// TIA Portal V20 export
FUNCTION_BLOCK "CallUnit"   // FB130, LAD
TITLE = CallUnit
// This block calls all functionality inside the unit.
// stored: IsIECCheckEnabled true, MemoryReserve 100, Namespace Unit1, SetENOAutomatically true
   VAR_INPUT
      safetyReleased : Bool;   // Status from safety program
   END_VAR
   VAR_OUTPUT
      acknowledgeSafety { ExternalWritable := 'False'} : Bool;   // Acknowledge command to the safety program
   END_VAR
   VAR_IN_OUT
      globalStatus : "LAF_typeGeneralStatus";   // Global status
      unitInterface : "LAF_typeUnitInterface";   // Global unit interface
   END_VAR
   VAR
      instManageAlarms { ExternalWritable := 'False'} : "LAF_ManageAlarms";
      instStatusCollector { ExternalWritable := 'False'} : "LUC_StatusCollector";
      instInterfaceManager { ExternalWritable := 'False'} : "LUC_InterfaceManager";
      instUnitModeStateManager { ExternalWritable := 'False'} : "LPMLV2022_UnitModeStateManager";
      instRemoteInterfaceOpcUa { ExternalWritable := 'False'} : "LUC_RemoteCtrl_OpcUa";
      instSignalStack { ExternalWritable := 'False'} : "LUC_SignalStack";
      instUnitModeStateTimes { ExternalWritable := 'False'} : "LPMLV2022_UnitModeStateTimes";
      instUnitModeChangeAllowed { ExternalWritable := 'False'} : "LPMLV2022_UnitModeChangeAllowed";
      instPFEEvents { ExternalWritable := 'False'} : "Unit1.EventsPFE";
      instTonTimer { ExternalWritable := 'False'} : Array[0..9] of TON_TIME;
      instTofTimer { ExternalWritable := 'False'} : Array[0..9] of TOF_TIME;
      instEQP_Interface_BA030 { ExternalWritable := 'False'} : "LER_EQP_Interface";
      instEQP_Interface_BA040 { ExternalWritable := 'False'} : "LER_EQP_Interface";
      instSinaInfeed { ExternalWritable := 'False'} : SinaInfeed;
      instLER_FFU_LIU117 { ExternalWritable := 'False'} : "LER_FFU_LIU117";
      statRemoteInterface { ExternalWritable := 'False'} : "LUC_typeCommands";
      statLocalInterface { ExternalWritable := 'False'} : "LUC_typeCommands";
      statEmEnableCheck { ExternalWritable := 'False'} : Array[0..2] of Bool;
      statEmHomedCheck { ExternalWritable := 'False'} : Array[0..2] of Bool;
      statPulse { ExternalWritable := 'False'} : Array[0..99] of Bool;
      statCycleTime { ExternalWritable := 'False'} : Struct
         Buffer1 : LReal;
         Buffer2 : DInt;
         Buffer3 : DInt;
         Buffer4 : DInt;
         Buffer5 : DInt;
      END_STRUCT;
      statEnableManualCmds : Bool;
      statAllEmLinked { ExternalWritable := 'False'} : Bool;
      citi_Ptrig : Array[0..20] of Bool;
      citiTon : Array[0..20] of TON_TIME;
      citi : Time;
      citiTest : Array[0..20] of Bool;
   END_VAR
   VAR_TEMP
      tempUnitFeedback : "LUC_typeStateCommands";   // Collected commands in the unit, e.g. direct command or commands derived from alarms
      tempProcessCommands : "LUC_typeStateCommands";   // Requested unit state changes by the process
      tempUnitMode : DInt;   // Requested unit mode
      tempUnitModeChangeRequest : Bool;   // Request unit mode
      tempCntrlCmd : DInt;   // Request control command
      tempCmdChangeRequest : Bool;   // Enable change into requested state
      tempSc : Bool;   // State change from FALSE to TRUE (rising edge) triggers state complete signal
      tempPartData : "LER_typePartData";
      tempPartData_All : Array[0..18] of "LER_typePartData";
      tempTimeMs : DInt;
   END_VAR
   VAR CONSTANT
      TRUE : Bool := TRUE;
      FALSE : Bool := FALSE;
   END_VAR
   VAR_TEMP   // added for the SCL form of the ladder/FBD networks
      _w1 : Bool;
      _w2 : Bool;
      _w3 : Bool;
      _w4 : Bool;
      _w5 : Bool;
      _w6 : Bool;
      _w7 : Bool;
      _w8 : Bool;
   END_VAR
BEGIN

REGION Network 1: BLOCK INFO HEADER
   // (company) / (C) Copyright (year)
   // ---------------------------------------------------------------------------------
   // Title:                             (Title of this block)
   // Comment/Function: (that is implemented in the block)
   // Library/Family:           (that the source is dedicated to)
   // Author:                        (department / person in charge / contact)
   // Target System:          (test system with FW version)
   // Engineering:              TIA Portal (SW version)
   // Restrictions:               (OB types, etc.)
   // Requirements:           (hardware, technological package, etc.)
   // ---------------------------------------------------------------------------------
   // Change log table:
   // Version          | Date             | Signature      | Expert in charge  | Changes applied ------------------------|----------------------|-------------------------|--------------------------------|-----------------------
   // 001.000.000 | yyyy-mm-dd | 0x00000000 | (name of expert) | First released version
END_REGION

REGION Network 2: DESCRIPTION
   // This is a template block provided by the Automation Framework. It can be used to create an own project.
   // The Block Info Header is prepared to put in your own data.
   // Description of the block could be added here and the docu created by Code2Docu.
END_REGION

REGION Network 3: Simulation
   // If simulation is active on a global level, inherit this status and set simulation active in this unit also. Information is written to DB ControlNodes, from where it is distributed to the equipmemt modules.
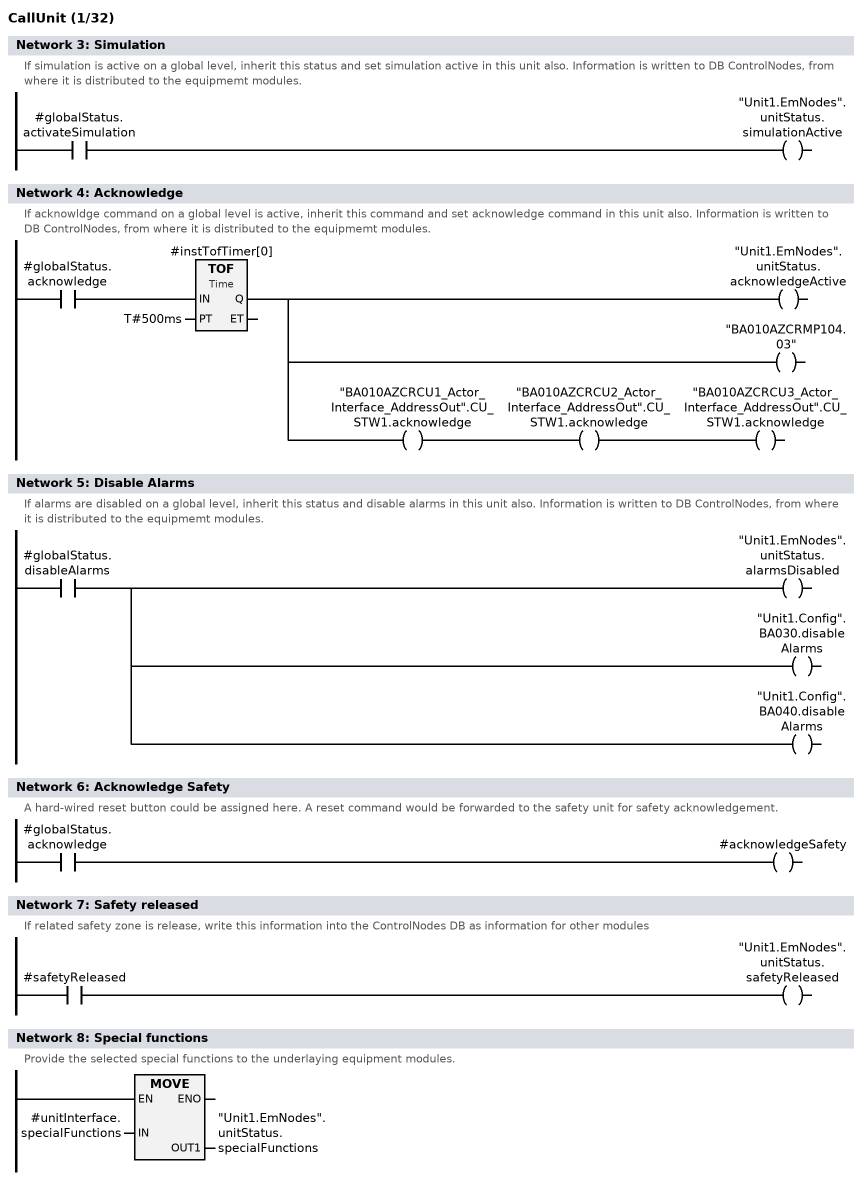
   RUNG wire#powerrail
      Contact( #globalStatus.activateSimulation )
      Coil( "Unit1.EmNodes".unitStatus.simulationActive )
   END_RUNG
   // the same network as SCL:
   "Unit1.EmNodes".unitStatus.simulationActive := #globalStatus.activateSimulation;
END_REGION

REGION Network 4: Acknowledge
   // If acknowldge command on a global level is active, inherit this command and set acknowledge command in this unit also. Information is written to DB ControlNodes, from where it is distributed to the equipmemt modules.
   RUNG wire#powerrail
      Contact( #globalStatus.acknowledge )
      { S7_Templates := "time_type := Time" } #instTofTimer[0].TOF(pt := T#500ms, et =>)
      wire#w1
      Coil( "Unit1.EmNodes".unitStatus.acknowledgeActive )
   END_RUNG
   RUNG wire#w1
      Coil( "BA010AZCRMP104.03" )
   END_RUNG
   RUNG wire#w1
      Coil( "BA010AZCRCU1_Actor_Interface_AddressOut".CU_STW1.acknowledge )
      Coil( "BA010AZCRCU2_Actor_Interface_AddressOut".CU_STW1.acknowledge )
      Coil( "BA010AZCRCU3_Actor_Interface_AddressOut".CU_STW1.acknowledge )
   END_RUNG
   // the same network as SCL:
   #instTofTimer[0].TOF(IN := #globalStatus.acknowledge, PT := T#500ms);
   "Unit1.EmNodes".unitStatus.acknowledgeActive := #instTofTimer[0].Q;
   "BA010AZCRMP104.03" := #instTofTimer[0].Q;
   "BA010AZCRCU1_Actor_Interface_AddressOut".CU_STW1.acknowledge := #instTofTimer[0].Q;
   "BA010AZCRCU2_Actor_Interface_AddressOut".CU_STW1.acknowledge := #instTofTimer[0].Q;
   "BA010AZCRCU3_Actor_Interface_AddressOut".CU_STW1.acknowledge := #instTofTimer[0].Q;
END_REGION

REGION Network 5: Disable Alarms
   // If alarms are disabled on a global level, inherit this status and disable alarms in this unit also. Information is written to DB ControlNodes, from where it is distributed to the equipmemt modules.
   RUNG wire#powerrail
      Contact( #globalStatus.disableAlarms )
      wire#w1
      Coil( "Unit1.EmNodes".unitStatus.alarmsDisabled )
   END_RUNG
   RUNG wire#w1
      Coil( "Unit1.Config".BA030.disableAlarms )
   END_RUNG
   RUNG wire#w1
      Coil( "Unit1.Config".BA040.disableAlarms )
   END_RUNG
   // the same network as SCL:
   "Unit1.EmNodes".unitStatus.alarmsDisabled := #globalStatus.disableAlarms;
   "Unit1.Config".BA030.disableAlarms := #globalStatus.disableAlarms;
   "Unit1.Config".BA040.disableAlarms := #globalStatus.disableAlarms;
END_REGION

REGION Network 6: Acknowledge Safety
   // A hard-wired reset button could be assigned here. A reset command would be forwarded to the safety unit for safety acknowledgement.
   RUNG wire#powerrail
      Contact( #globalStatus.acknowledge )
      Coil( #acknowledgeSafety )
   END_RUNG
   // the same network as SCL:
   #acknowledgeSafety := #globalStatus.acknowledge;
END_REGION

REGION Network 7: Safety released
   // If related safety zone is release, write this information into the ControlNodes DB as information for other modules
   RUNG wire#powerrail
      Contact( #safetyReleased )
      Coil( "Unit1.EmNodes".unitStatus.safetyReleased )
   END_RUNG
   // the same network as SCL:
   "Unit1.EmNodes".unitStatus.safetyReleased := #safetyReleased;
END_REGION

REGION Network 8: Special functions
   // Provide the selected special functions to the underlaying equipment modules.
   RUNG wire#powerrail
      Move(in := #unitInterface.specialFunctions, out1 => "Unit1.EmNodes".unitStatus.specialFunctions)
   END_RUNG
   // the same network as SCL:
   "Unit1.EmNodes".unitStatus.specialFunctions := #unitInterface.specialFunctions;
END_REGION

REGION Network 9 (SCL): Electric Power CB
   // E.g. put the feedback of circuit breakers or power supplies here.
   // DC24 Voltage
   "Unit1.ControlNodes".fuses.E726CbVoltage24VOK := "BA010AZCRMP101.12";
   "Unit1.ControlNodes".fuses.E4304CbVoltage24VOK := "BA010AZCRMP101.17";
   "Unit1.ControlNodes".fuses.E4420CbVoltage24VOK := "BA010AZCRMP101.22";
   "Unit1.ControlNodes".fuses.E4426CbVoltage24VOK := "BA010AZCRMP101.23";
   "Unit1.ControlNodes".fuses.E4432CbVoltage24VOK := "BA010AZCRMP101.24";
   "Unit1.ControlNodes".fuses.E4456CbVoltage24VOK := "BA010AZCRMP101.25";
   "Unit1.ControlNodes".fuses.E5110CbVoltage24VOK := "BA010AZCRMP101.31";
   "Unit1.ControlNodes".fuses.E5116CbVoltage24VOK := "BA010AZCRMP101.32";
   "Unit1.ControlNodes".fuses.E5160CbVoltage24VOK := "BA010AZCRMP101.33";
   "Unit1.ControlNodes".fuses.E5166CbVoltage24VOK := "BA010AZCRMP101.34";
   "Unit1.ControlNodes".fuses.E5172CbVoltage24VOK := "BA010AZCRMP101.35";
   "Unit1.ControlNodes".fuses.E5222CbVoltage24VOK := "BA010AZCRMP101.37";
   "Unit1.ControlNodes".fuses.E6154CbVoltage24VOK := "BA010AZCRMP102.02";
   "Unit1.ControlNodes".fuses.E6180CbVoltage24VOK := "BA010AZCRMP102.03";
   "Unit1.ControlNodes".fuses.E6204CbVoltage24VOK := "BA010AZCRMP102.04";
   "Unit1.ControlNodes".fuses.E6206CbVoltage24VOK := "BA010AZCRMP102.05";
   "Unit1.ControlNodes".fuses.E6220CbVoltage24VOK := "BA010AZCRMP102.06";
   "Unit1.ControlNodes".fuses.E6224CbVoltage24VOK := "BA010AZCRMP102.07";
   "Unit1.ControlNodes".fuses.E6228CbVoltage24VOK := "BA010AZCRMP102.10";
   "Unit1.ControlNodes".fuses.E6304CbVoltage24VOK := "BA010AZCRMP102.12";
   "Unit1.ControlNodes".fuses.E6406CbVoltage24VOK := "BA010AZCRMP102.15";
   "Unit1.ControlNodes".fuses.E6416CbVoltage24VOK := "BA010AZCRMP102.16";
   "Unit1.ControlNodes".fuses.E6422CbVoltage24VOK := "BA010AZCRMP102.17";
   "Unit1.ControlNodes".fuses.E6456CbVoltage24VOK := "BA010AZCRMP102.21";
   "Unit1.ControlNodes".fuses.E6462CbVoltage24VOK := "BA010AZCRMP102.22";
   "Unit1.ControlNodes".fuses.E6468CbVoltage24VOK := "BA010AZCRMP102.23";
   "Unit1.ControlNodes".fuses.E6706CbVoltage24VOK := "BA010AZCRMP102.27";
   "Unit1.ControlNodes".fuses.E6716CbVoltage24VOK := "BA010AZCRMP102.30";
   "Unit1.ControlNodes".fuses.E6722CbVoltage24VOK := "BA010AZCRMP102.31";
   "Unit1.ControlNodes".fuses.E6728CbVoltage24VOK := "BA010AZCRMP102.32";
   "Unit1.ControlNodes".fuses.E6734CbVoltage24VOK := "BA010AZCRMP102.33";
   "Unit1.ControlNodes".fuses.E6756CbVoltage24VOK := "BA010AZCRMP102.34";
   "Unit1.ControlNodes".fuses.E6762CbVoltage24VOK := "BA010AZCRMP102.35";
   "Unit1.ControlNodes".fuses.E6768CbVoltage24VOK := "BA010AZCRMP102.36";
   "Unit1.ControlNodes".fuses.E6774CbVoltage24VOK := "BA010AZCRMP102.37";
   "Unit1.ControlNodes".fuses.E6780CbVoltage24VOK := "BA010AZCRMP103.00";
   "Unit1.ControlNodes".fuses.E6786CbVoltage24VOK := "BA010AZCRMP103.01";
   "Unit1.ControlNodes".fuses.E6806CbVoltage24VOK := "BA010AZCRMP103.03";
   "Unit1.ControlNodes".fuses.E6816CbVoltage24VOK := "BA010AZCRMP103.04";
   "Unit1.ControlNodes".fuses.E6836CbVoltage24VOK := "BA010AZCRMP103.05";
   "Unit1.ControlNodes".fuses.E6856CbVoltage24VOK := "BA010AZCRMP103.06";
   "Unit1.ControlNodes".fuses.E110CbVoltage24VOK := "BA010AZCRSP201.10";
   "Unit1.ControlNodes".fuses.E156CbVoltage24VOK := "BA010AZCRSP501.00";
   "Unit1.ControlNodes".fuses.E218CbVoltage24VOK := "BA010AZCRSP501.01";

   // AC480 Voltage
   "Unit1.ControlNodes".fuses.E202Cb480vVoltage24VOK := "BA010AZCRMP101.00";
   "Unit1.ControlNodes".fuses.E208Cb480vVoltage24VOK := "BA010AZCRMP101.01";
   "Unit1.ControlNodes".fuses.E214Cb480vVoltage24VOK := "BA010AZCRMP101.02";
   "Unit1.ControlNodes".fuses.E220Cb480vVoltage24VOK := "BA010AZCRMP101.03";
   "Unit1.ControlNodes".fuses.E320Cb480vVoltage24VOK := "BA010AZCRMP101.05";
   "Unit1.ControlNodes".fuses.E326Cb480vVoltage24VOK := "BA010AZCRMP101.06";
   "Unit1.ControlNodes".fuses.E332Cb480vVoltage24VOK := "BA010AZCRMP101.07";
   "Unit1.ControlNodes".fuses.E720Cb480vVoltage24VOK := "BA010AZCRMP101.11";
   "Unit1.ControlNodes".fuses.E4116Cb480vVoltage24VOK := "BA010AZCRMP101.14";
   "Unit1.ControlNodes".fuses.E4156Cb480vVoltage24VOK := "BA010AZCRMP101.15";
   "Unit1.ControlNodes".fuses.E5100Cb480vVoltage24VOK := "BA010AZCRMP101.30";
END_REGION

REGION Network 10 (SCL): Power Supply
   "Unit1.ControlNodes".pws.powerSupplyE4404PwsOK := "BA010AZCRMP101.21";
   "Unit1.ControlNodes".pws.powerSupplyE6104PwsOK := "BA010AZCRMP102.01";
   "Unit1.ControlNodes".pws.powerSupplyE6404PwsOK := "BA010AZCRMP102.14";
   "Unit1.ControlNodes".pws.powerSupplyE6704PwsOK := "BA010AZCRMP102.26";
   "Unit1.ControlNodes".pws.powerSupplyE6804PwsOK := "BA010AZCRMP103.02";
END_REGION

REGION Network 11: Main Air OK
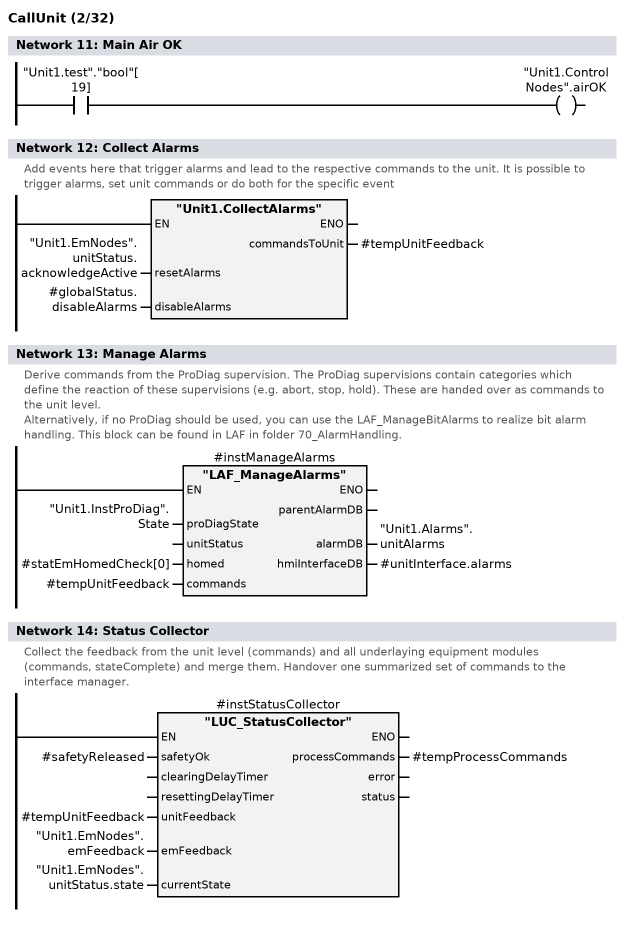
   RUNG wire#powerrail
      Contact( "Unit1.test"."bool"[19] )
      Coil( "Unit1.ControlNodes".airOK )
   END_RUNG
   // the same network as SCL:
   "Unit1.ControlNodes".airOK := "Unit1.test"."bool"[19];
END_REGION

REGION Network 12: Collect Alarms
   // Add events here that trigger alarms and lead to the respective commands to the unit. It is possible to trigger alarms, set unit commands or do both for the specific event
   RUNG wire#powerrail
      "Unit1.CollectAlarms"(resetAlarms := "Unit1.EmNodes".unitStatus.acknowledgeActive, disableAlarms := #globalStatus.disableAlarms, commandsToUnit => #tempUnitFeedback)
   END_RUNG
   // the same network as SCL:
   "Unit1.CollectAlarms"(resetAlarms := "Unit1.EmNodes".unitStatus.acknowledgeActive,
                         disableAlarms := #globalStatus.disableAlarms,
                         commandsToUnit => #tempUnitFeedback);
END_REGION

REGION Network 13: Manage Alarms
   // Derive commands from the ProDiag supervision. The ProDiag supervisions contain categories which define the reaction of these supervisions (e.g. abort, stop, hold). These are handed over as commands to the unit level.
   // Alternatively, if no ProDiag should be used, you can use the LAF_ManageBitAlarms to realize bit alarm handling. This block can be found in LAF in folder 70_AlarmHandling.
   RUNG wire#powerrail
      #instManageAlarms(proDiagState := "Unit1.InstProDiag".State, unitStatus :=, homed := #statEmHomedCheck[0], commands := #tempUnitFeedback, parentAlarmDB =>, alarmDB => "Unit1.Alarms".unitAlarms, hmiInterfaceDB => #unitInterface.alarms)
   END_RUNG
   // the same network as SCL:
   #instManageAlarms(proDiagState := "Unit1.InstProDiag".State,   // "LAF_ManageAlarms"
                     homed := #statEmHomedCheck[0],
                     commands := #tempUnitFeedback,
                     alarmDB => "Unit1.Alarms".unitAlarms,
                     hmiInterfaceDB => #unitInterface.alarms);
END_REGION

REGION Network 14: Status Collector
   // Collect the feedback from the unit level (commands) and all underlaying equipment modules (commands, stateComplete) and merge them. Handover one summarized set of commands to the interface manager.
   RUNG wire#powerrail
      #instStatusCollector(safetyOk := #safetyReleased, clearingDelayTimer :=, resettingDelayTimer :=, unitFeedback := #tempUnitFeedback, emFeedback := "Unit1.EmNodes".emFeedback, currentState := "Unit1.EmNodes".unitStatus.state, processCommands => #tempProcessCommands, error =>, status =>)
   END_RUNG
   // the same network as SCL:
   #instStatusCollector(safetyOk := #safetyReleased,   // "LUC_StatusCollector"
                        unitFeedback := #tempUnitFeedback,
                        emFeedback := "Unit1.EmNodes".emFeedback,
                        currentState := "Unit1.EmNodes".unitStatus.state,
                        processCommands => #tempProcessCommands);
END_REGION

REGION Network 15: Interface Manager
   // Read the commands from all interfaces (process, local, hmi, remote) and merge them. Handover one summarized set of commands to the mode state manager.
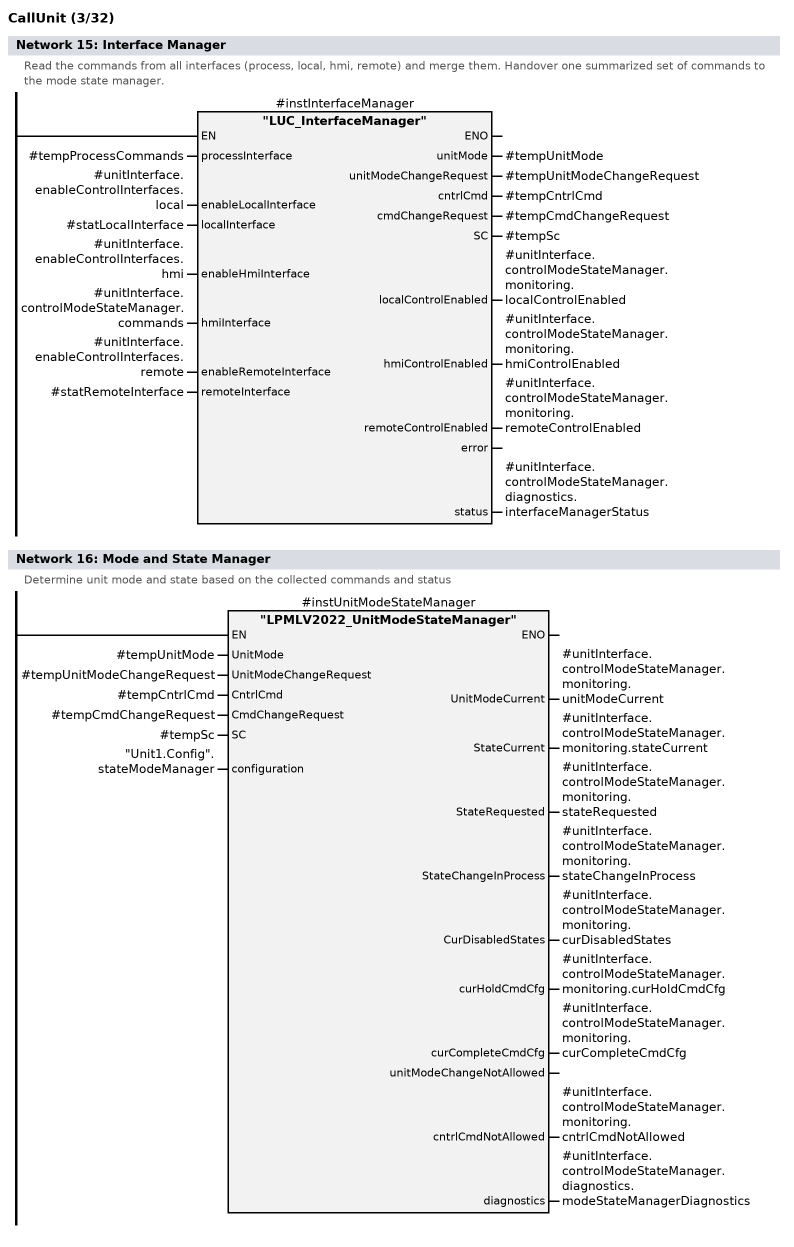
   RUNG wire#powerrail
      #instInterfaceManager(processInterface := #tempProcessCommands, enableLocalInterface := #unitInterface.enableControlInterfaces.local, localInterface := #statLocalInterface, enableHmiInterface := #unitInterface.enableControlInterfaces.hmi, hmiInterface := #unitInterface.controlModeStateManager.commands, enableRemoteInterface := #unitInterface.enableControlInterfaces.remote, remoteInterface := #statRemoteInterface, unitMode => #tempUnitMode, unitModeChangeRequest => #tempUnitModeChangeRequest, cntrlCmd => #tempCntrlCmd, cmdChangeRequest => #tempCmdChangeRequest, SC => #tempSc, localControlEnabled => #unitInterface.controlModeStateManager.monitoring.localControlEnabled, hmiControlEnabled => #unitInterface.controlModeStateManager.monitoring.hmiControlEnabled, remoteControlEnabled => #unitInterface.controlModeStateManager.monitoring.remoteControlEnabled, error =>, status => #unitInterface.controlModeStateManager.diagnostics.interfaceManagerStatus)
   END_RUNG
   // the same network as SCL:
   #instInterfaceManager(processInterface := #tempProcessCommands,   // "LUC_InterfaceManager"
                         enableLocalInterface := #unitInterface.enableControlInterfaces.local,
                         localInterface := #statLocalInterface,
                         enableHmiInterface := #unitInterface.enableControlInterfaces.hmi,
                         hmiInterface := #unitInterface.controlModeStateManager.commands,
                         enableRemoteInterface := #unitInterface.enableControlInterfaces.remote,
                         remoteInterface := #statRemoteInterface,
                         unitMode => #tempUnitMode,
                         unitModeChangeRequest => #tempUnitModeChangeRequest,
                         cntrlCmd => #tempCntrlCmd,
                         cmdChangeRequest => #tempCmdChangeRequest,
                         SC => #tempSc,
                         localControlEnabled => #unitInterface.controlModeStateManager.monitoring.localControlEnabled,
                         hmiControlEnabled => #unitInterface.controlModeStateManager.monitoring.hmiControlEnabled,
                         remoteControlEnabled => #unitInterface.controlModeStateManager.monitoring.remoteControlEnabled,
                         status => #unitInterface.controlModeStateManager.diagnostics.interfaceManagerStatus);
END_REGION

REGION Network 16: Mode and State Manager
   // Determine unit mode and state based on the collected commands and status
   RUNG wire#powerrail
      #instUnitModeStateManager(UnitMode := #tempUnitMode, UnitModeChangeRequest := #tempUnitModeChangeRequest, CntrlCmd := #tempCntrlCmd, CmdChangeRequest := #tempCmdChangeRequest, SC := #tempSc, configuration := "Unit1.Config".stateModeManager, UnitModeCurrent => #unitInterface.controlModeStateManager.monitoring.unitModeCurrent, StateCurrent => #unitInterface.controlModeStateManager.monitoring.stateCurrent, StateRequested => #unitInterface.controlModeStateManager.monitoring.stateRequested, StateChangeInProcess => #unitInterface.controlModeStateManager.monitoring.stateChangeInProcess, CurDisabledStates => #unitInterface.controlModeStateManager.monitoring.curDisabledStates, curHoldCmdCfg => #unitInterface.controlModeStateManager.monitoring.curHoldCmdCfg, curCompleteCmdCfg => #unitInterface.controlModeStateManager.monitoring.curCompleteCmdCfg, unitModeChangeNotAllowed =>, cntrlCmdNotAllowed => #unitInterface.controlModeStateManager.monitoring.cntrlCmdNotAllowed, diagnostics => #unitInterface.controlModeStateManager.diagnostics.modeStateManagerDiagnostics)
   END_RUNG
   // the same network as SCL:
   #instUnitModeStateManager(UnitMode := #tempUnitMode,   // "LPMLV2022_UnitModeStateManager"
                           UnitModeChangeRequest := #tempUnitModeChangeRequest,
                           CntrlCmd := #tempCntrlCmd,
                           CmdChangeRequest := #tempCmdChangeRequest,
                           SC := #tempSc,
                           configuration := "Unit1.Config".stateModeManager,
                           UnitModeCurrent => #unitInterface.controlModeStateManager.monitoring.unitModeCurrent,
                           StateCurrent => #unitInterface.controlModeStateManager.monitoring.stateCurrent,
                           StateRequested => #unitInterface.controlModeStateManager.monitoring.stateRequested,
                           StateChangeInProcess => #unitInterface.controlModeStateManager.monitoring.stateChangeInProcess,
                           CurDisabledStates => #unitInterface.controlModeStateManager.monitoring.curDisabledStates,
                           curHoldCmdCfg => #unitInterface.controlModeStateManager.monitoring.curHoldCmdCfg,
                           curCompleteCmdCfg => #unitInterface.controlModeStateManager.monitoring.curCompleteCmdCfg,
                           cntrlCmdNotAllowed => #unitInterface.controlModeStateManager.monitoring.cntrlCmdNotAllowed,
                           diagnostics => #unitInterface.controlModeStateManager.diagnostics.modeStateManagerDiagnostics);
END_REGION

REGION Network 17: Helper Functions
   // 1. Read mode and state from the mode state manager an write them to the DB ControlNode
   // 2. Read mode and state from the mode state manager, translate them to a string and write them in unitInterface
   // 3. Determine if a mode change is allowed in the current state and write that information to the unitInterface
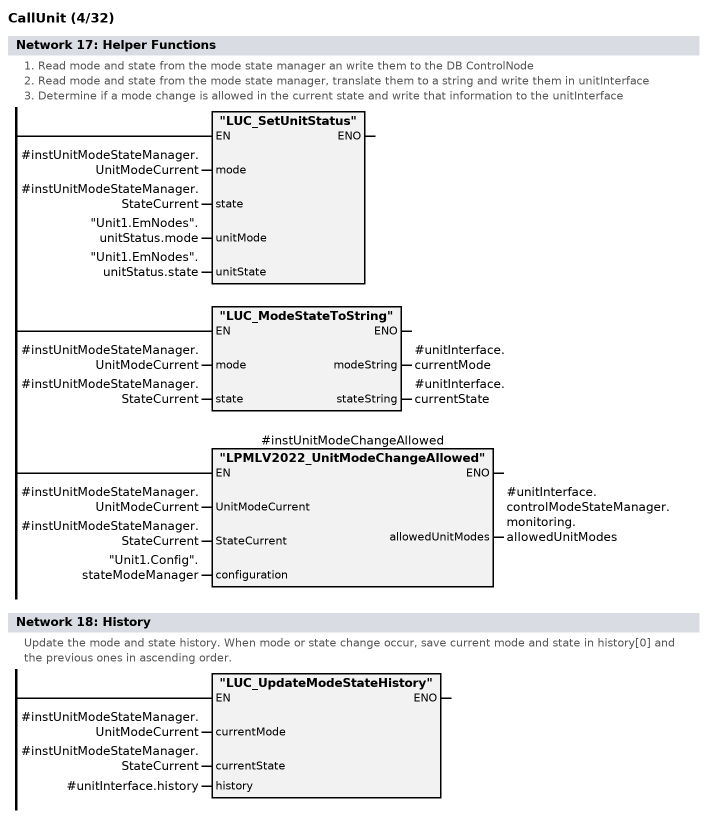
   RUNG wire#powerrail
      "LUC_SetUnitStatus"(mode := #instUnitModeStateManager.UnitModeCurrent, state := #instUnitModeStateManager.StateCurrent, unitMode := "Unit1.EmNodes".unitStatus.mode, unitState := "Unit1.EmNodes".unitStatus.state)
   END_RUNG
   RUNG wire#powerrail
      "LUC_ModeStateToString"(mode := #instUnitModeStateManager.UnitModeCurrent, state := #instUnitModeStateManager.StateCurrent, modeString => #unitInterface.currentMode, stateString => #unitInterface.currentState)
   END_RUNG
   RUNG wire#powerrail
      #instUnitModeChangeAllowed(UnitModeCurrent := #instUnitModeStateManager.UnitModeCurrent, StateCurrent := #instUnitModeStateManager.StateCurrent, configuration := "Unit1.Config".stateModeManager, allowedUnitModes => #unitInterface.controlModeStateManager.monitoring.allowedUnitModes)
   END_RUNG
   // the same network as SCL:
   "LUC_SetUnitStatus"(mode := #instUnitModeStateManager.UnitModeCurrent,
                       state := #instUnitModeStateManager.StateCurrent,
                       unitMode := "Unit1.EmNodes".unitStatus.mode,
                       unitState := "Unit1.EmNodes".unitStatus.state);
   "LUC_ModeStateToString"(mode := #instUnitModeStateManager.UnitModeCurrent,
                           state := #instUnitModeStateManager.StateCurrent,
                           modeString => #unitInterface.currentMode,
                           stateString => #unitInterface.currentState);
   #instUnitModeChangeAllowed(UnitModeCurrent := #instUnitModeStateManager.UnitModeCurrent,   // "LPMLV2022_UnitModeChangeAllowed"
                           StateCurrent := #instUnitModeStateManager.StateCurrent,
                           configuration := "Unit1.Config".stateModeManager,
                           allowedUnitModes => #unitInterface.controlModeStateManager.monitoring.allowedUnitModes);
END_REGION

REGION Network 18: History
   // Update the mode and state history. When mode or state change occur, save current mode and state in history[0] and the previous ones in ascending order.
   RUNG wire#powerrail
      "LUC_UpdateModeStateHistory"(currentMode := #instUnitModeStateManager.UnitModeCurrent, currentState := #instUnitModeStateManager.StateCurrent, history := #unitInterface.history)
   END_RUNG
   // the same network as SCL:
   "LUC_UpdateModeStateHistory"(currentMode := #instUnitModeStateManager.UnitModeCurrent,
                           currentState := #instUnitModeStateManager.StateCurrent,
                           history := #unitInterface.history);
END_REGION

REGION Network 19: Time Statistics
   // Determine the time that has been spend in modes and states.
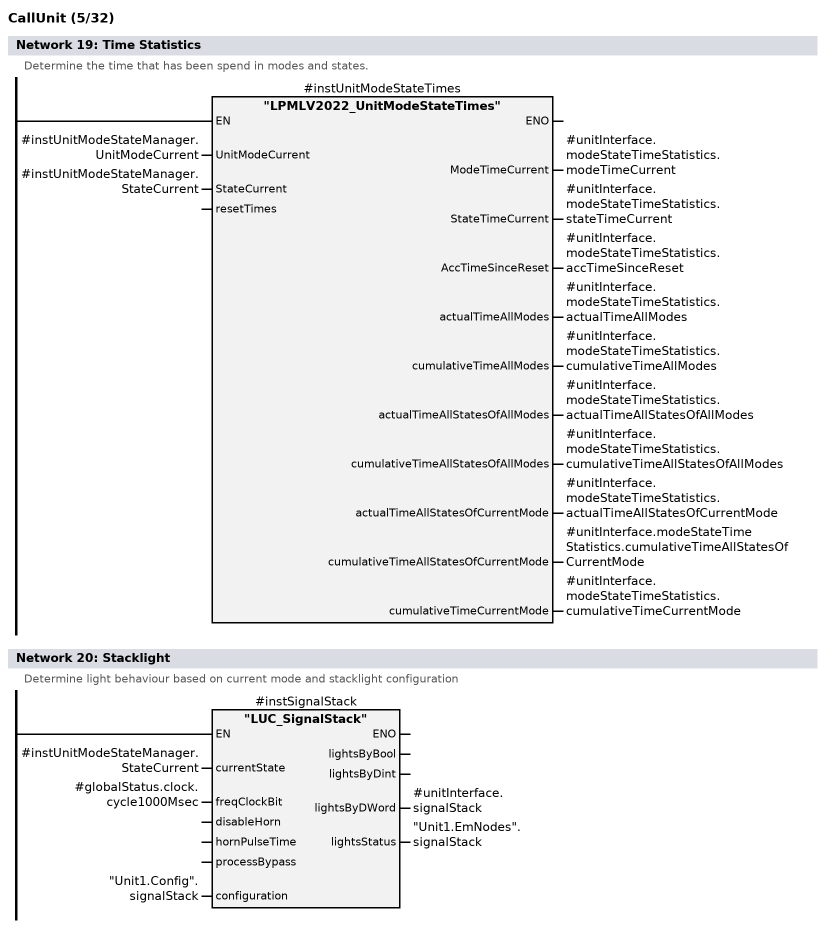
   RUNG wire#powerrail
      #instUnitModeStateTimes(UnitModeCurrent := #instUnitModeStateManager.UnitModeCurrent, StateCurrent := #instUnitModeStateManager.StateCurrent, resetTimes :=, ModeTimeCurrent => #unitInterface.modeStateTimeStatistics.modeTimeCurrent, StateTimeCurrent => #unitInterface.modeStateTimeStatistics.stateTimeCurrent, AccTimeSinceReset => #unitInterface.modeStateTimeStatistics.accTimeSinceReset, actualTimeAllModes => #unitInterface.modeStateTimeStatistics.actualTimeAllModes, cumulativeTimeAllModes => #unitInterface.modeStateTimeStatistics.cumulativeTimeAllModes, actualTimeAllStatesOfAllModes => #unitInterface.modeStateTimeStatistics.actualTimeAllStatesOfAllModes, cumulativeTimeAllStatesOfAllModes => #unitInterface.modeStateTimeStatistics.cumulativeTimeAllStatesOfAllModes, actualTimeAllStatesOfCurrentMode => #unitInterface.modeStateTimeStatistics.actualTimeAllStatesOfCurrentMode, cumulativeTimeAllStatesOfCurrentMode => #unitInterface.modeStateTimeStatistics.cumulativeTimeAllStatesOfCurrentMode, cumulativeTimeCurrentMode => #unitInterface.modeStateTimeStatistics.cumulativeTimeCurrentMode)
   END_RUNG
   // the same network as SCL:
   #instUnitModeStateTimes(UnitModeCurrent := #instUnitModeStateManager.UnitModeCurrent,   // "LPMLV2022_UnitModeStateTimes"
                           StateCurrent := #instUnitModeStateManager.StateCurrent,
                           ModeTimeCurrent => #unitInterface.modeStateTimeStatistics.modeTimeCurrent,
                           StateTimeCurrent => #unitInterface.modeStateTimeStatistics.stateTimeCurrent,
                           AccTimeSinceReset => #unitInterface.modeStateTimeStatistics.accTimeSinceReset,
                           actualTimeAllModes => #unitInterface.modeStateTimeStatistics.actualTimeAllModes,
                           cumulativeTimeAllModes => #unitInterface.modeStateTimeStatistics.cumulativeTimeAllModes,
                           actualTimeAllStatesOfAllModes => #unitInterface.modeStateTimeStatistics.actualTimeAllStatesOfAllModes,
                           cumulativeTimeAllStatesOfAllModes => #unitInterface.modeStateTimeStatistics.cumulativeTimeAllStatesOfAllModes,
                           actualTimeAllStatesOfCurrentMode => #unitInterface.modeStateTimeStatistics.actualTimeAllStatesOfCurrentMode,
                           cumulativeTimeAllStatesOfCurrentMode => #unitInterface.modeStateTimeStatistics.cumulativeTimeAllStatesOfCurrentMode,
                           cumulativeTimeCurrentMode => #unitInterface.modeStateTimeStatistics.cumulativeTimeCurrentMode);
END_REGION

REGION Network 20: Stacklight
   // Determine light behaviour based on current mode and stacklight configuration
   RUNG wire#powerrail
      #instSignalStack(currentState := #instUnitModeStateManager.StateCurrent, freqClockBit := #globalStatus.clock.cycle1000Msec, disableHorn :=, hornPulseTime :=, processBypass :=, configuration := "Unit1.Config".signalStack, lightsByBool =>, lightsByDint =>, lightsByDWord => #unitInterface.signalStack, lightsStatus => "Unit1.EmNodes".signalStack)
   END_RUNG
   // the same network as SCL:
   #instSignalStack(currentState := #instUnitModeStateManager.StateCurrent,   // "LUC_SignalStack"
                    freqClockBit := #globalStatus.clock.cycle1000Msec,
                    configuration := "Unit1.Config".signalStack,
                    lightsByDWord => #unitInterface.signalStack,
                    lightsStatus => "Unit1.EmNodes".signalStack);
END_REGION

REGION Network 21: Stacklight Lamp
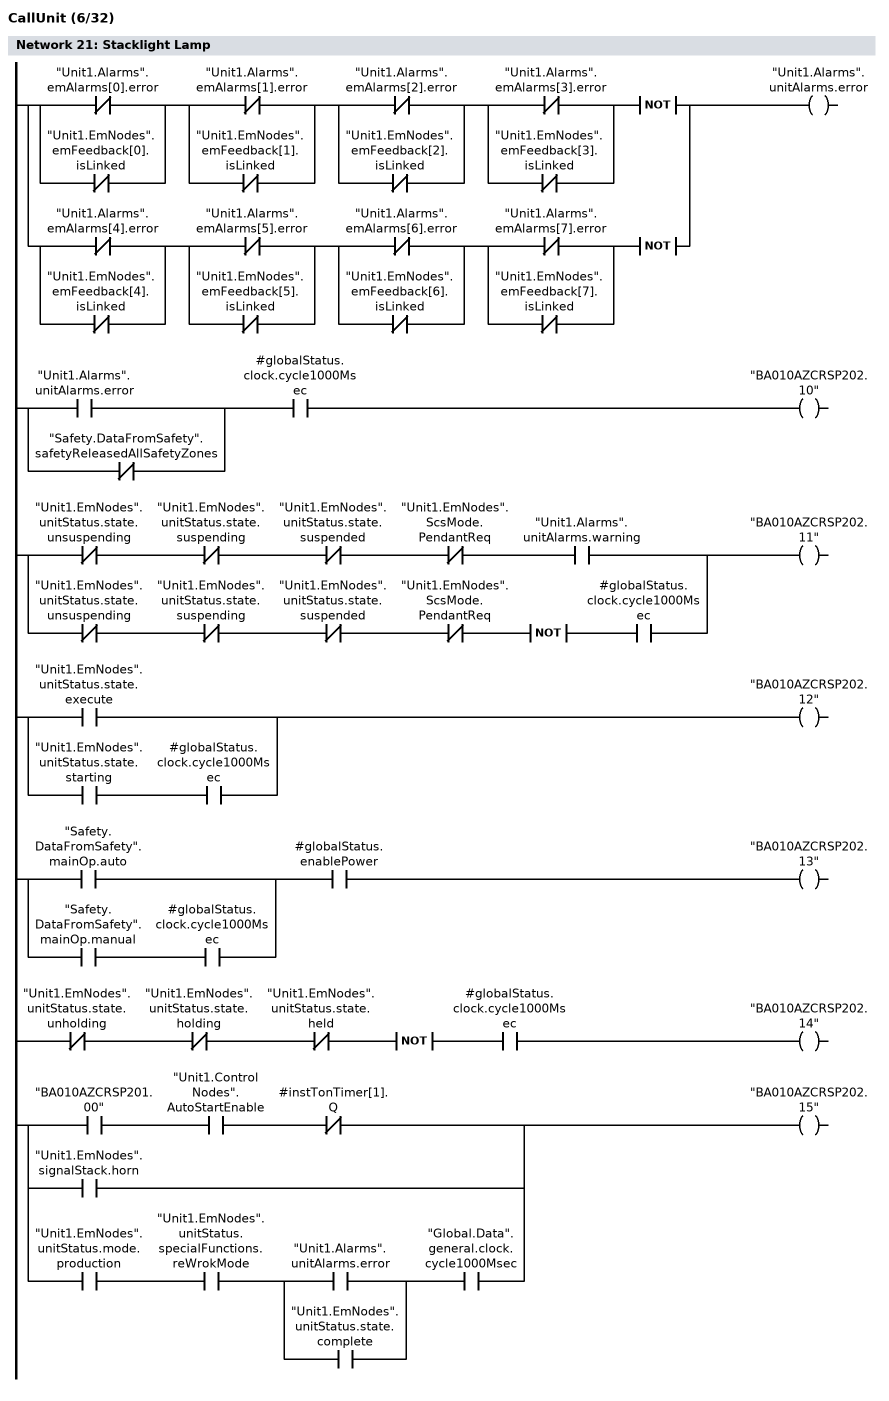
   RUNG wire#powerrail
      I_Contact( "Unit1.Alarms".emAlarms[0].error )
      wire#w1
      I_Contact( "Unit1.Alarms".emAlarms[1].error )
      wire#w2
      I_Contact( "Unit1.Alarms".emAlarms[2].error )
      wire#w3
      I_Contact( "Unit1.Alarms".emAlarms[3].error )
      wire#w4
      Not()
      wire#w5
      Coil( "Unit1.Alarms".unitAlarms.error )
   END_RUNG
   RUNG wire#powerrail
      I_Contact( "Unit1.EmNodes".emFeedback[0].isLinked )
   END_RUNG wire#w1
   RUNG wire#w1
      I_Contact( "Unit1.EmNodes".emFeedback[1].isLinked )
   END_RUNG wire#w2
   RUNG wire#w2
      I_Contact( "Unit1.EmNodes".emFeedback[2].isLinked )
   END_RUNG wire#w3
   RUNG wire#w3
      I_Contact( "Unit1.EmNodes".emFeedback[3].isLinked )
   END_RUNG wire#w4
   RUNG wire#powerrail
      I_Contact( "Unit1.Alarms".emAlarms[4].error )
      wire#w6
      I_Contact( "Unit1.Alarms".emAlarms[5].error )
      wire#w7
      I_Contact( "Unit1.Alarms".emAlarms[6].error )
      wire#w8
      I_Contact( "Unit1.Alarms".emAlarms[7].error )
      wire#w9
      Not()
   END_RUNG wire#w5
   RUNG wire#powerrail
      I_Contact( "Unit1.EmNodes".emFeedback[4].isLinked )
   END_RUNG wire#w6
   RUNG wire#w6
      I_Contact( "Unit1.EmNodes".emFeedback[5].isLinked )
   END_RUNG wire#w7
   RUNG wire#w7
      I_Contact( "Unit1.EmNodes".emFeedback[6].isLinked )
   END_RUNG wire#w8
   RUNG wire#w8
      I_Contact( "Unit1.EmNodes".emFeedback[7].isLinked )
   END_RUNG wire#w9
   RUNG wire#powerrail
      Contact( "Unit1.Alarms".unitAlarms.error )
      wire#w10
      Contact( #globalStatus.clock.cycle1000Msec )
      Coil( "BA010AZCRSP202.10" )
   END_RUNG
   RUNG wire#powerrail
      I_Contact( "Safety.DataFromSafety".safetyReleasedAllSafetyZones )
   END_RUNG wire#w10
   RUNG wire#powerrail
      I_Contact( "Unit1.EmNodes".unitStatus.state.unsuspending )
      I_Contact( "Unit1.EmNodes".unitStatus.state.suspending )
      I_Contact( "Unit1.EmNodes".unitStatus.state.suspended )
      I_Contact( "Unit1.EmNodes".ScsMode.PendantReq )
      Contact( "Unit1.Alarms".unitAlarms.warning )
      wire#w11
      Coil( "BA010AZCRSP202.11" )
   END_RUNG
   RUNG wire#powerrail
      I_Contact( "Unit1.EmNodes".unitStatus.state.unsuspending )
      I_Contact( "Unit1.EmNodes".unitStatus.state.suspending )
      I_Contact( "Unit1.EmNodes".unitStatus.state.suspended )
      I_Contact( "Unit1.EmNodes".ScsMode.PendantReq )
      Not()
      Contact( #globalStatus.clock.cycle1000Msec )
   END_RUNG wire#w11
   RUNG wire#powerrail
      Contact( "Unit1.EmNodes".unitStatus.state.execute )
      wire#w12
      Coil( "BA010AZCRSP202.12" )
   END_RUNG
   RUNG wire#powerrail
      Contact( "Unit1.EmNodes".unitStatus.state.starting )
      Contact( #globalStatus.clock.cycle1000Msec )
   END_RUNG wire#w12
   RUNG wire#powerrail
      Contact( "Safety.DataFromSafety".mainOp.auto )
      wire#w13
      Contact( #globalStatus.enablePower )
      Coil( "BA010AZCRSP202.13" )
   END_RUNG
   RUNG wire#powerrail
      Contact( "Safety.DataFromSafety".mainOp.manual )
      Contact( #globalStatus.clock.cycle1000Msec )
   END_RUNG wire#w13
   RUNG wire#powerrail
      I_Contact( "Unit1.EmNodes".unitStatus.state.unholding )
      I_Contact( "Unit1.EmNodes".unitStatus.state.holding )
      I_Contact( "Unit1.EmNodes".unitStatus.state.held )
      Not()
      Contact( #globalStatus.clock.cycle1000Msec )
      Coil( "BA010AZCRSP202.14" )
   END_RUNG
   RUNG wire#powerrail
      Contact( "BA010AZCRSP201.00" )
      Contact( "Unit1.ControlNodes".AutoStartEnable )
      I_Contact( #instTonTimer[1].Q )
      wire#w14
      Coil( "BA010AZCRSP202.15" )
   END_RUNG
   RUNG wire#powerrail
      Contact( "Unit1.EmNodes".signalStack.horn )
   END_RUNG wire#w14
   RUNG wire#powerrail
      Contact( "Unit1.EmNodes".unitStatus.mode.production )
      Contact( "Unit1.EmNodes".unitStatus.specialFunctions.reWrokMode )
      wire#w15
      Contact( "Unit1.Alarms".unitAlarms.error )
      wire#w16
      Contact( "Global.Data".general.clock.cycle1000Msec )
   END_RUNG wire#w14
   RUNG wire#w15
      Contact( "Unit1.EmNodes".unitStatus.state.complete )
   END_RUNG wire#w16
   // the same network as SCL:
   "Unit1.Alarms".unitAlarms.error := NOT ((NOT "Unit1.Alarms".emAlarms[0].error OR NOT "Unit1.EmNodes".emFeedback[0].isLinked) AND (NOT "Unit1.Alarms".emAlarms[1].error OR NOT "Unit1.EmNodes".emFeedback[1].isLinked) AND (NOT "Unit1.Alarms".emAlarms[2].error OR NOT "Unit1.EmNodes".emFeedback[2].isLinked) AND (NOT "Unit1.Alarms".emAlarms[3].error OR NOT "Unit1.EmNodes".emFeedback[3].isLinked)) OR NOT ((NOT "Unit1.Alarms".emAlarms[4].error OR NOT "Unit1.EmNodes".emFeedback[4].isLinked) AND (NOT "Unit1.Alarms".emAlarms[5].error OR NOT "Unit1.EmNodes".emFeedback[5].isLinked) AND (NOT "Unit1.Alarms".emAlarms[6].error OR NOT "Unit1.EmNodes".emFeedback[6].isLinked) AND (NOT "Unit1.Alarms".emAlarms[7].error OR NOT "Unit1.EmNodes".emFeedback[7].isLinked));
   "BA010AZCRSP202.10" := ("Unit1.Alarms".unitAlarms.error OR NOT "Safety.DataFromSafety".safetyReleasedAllSafetyZones) AND #globalStatus.clock.cycle1000Msec;
   "BA010AZCRSP202.11" := (NOT "Unit1.EmNodes".unitStatus.state.unsuspending AND NOT "Unit1.EmNodes".unitStatus.state.suspending AND NOT "Unit1.EmNodes".unitStatus.state.suspended AND NOT "Unit1.EmNodes".ScsMode.PendantReq AND "Unit1.Alarms".unitAlarms.warning) OR (NOT (NOT "Unit1.EmNodes".unitStatus.state.unsuspending AND NOT "Unit1.EmNodes".unitStatus.state.suspending AND NOT "Unit1.EmNodes".unitStatus.state.suspended AND NOT "Unit1.EmNodes".ScsMode.PendantReq) AND #globalStatus.clock.cycle1000Msec);
   "BA010AZCRSP202.12" := "Unit1.EmNodes".unitStatus.state.execute OR ("Unit1.EmNodes".unitStatus.state.starting AND #globalStatus.clock.cycle1000Msec);
   "BA010AZCRSP202.13" := ("Safety.DataFromSafety".mainOp.auto OR ("Safety.DataFromSafety".mainOp.manual AND #globalStatus.clock.cycle1000Msec)) AND #globalStatus.enablePower;
   "BA010AZCRSP202.14" := NOT (NOT "Unit1.EmNodes".unitStatus.state.unholding AND NOT "Unit1.EmNodes".unitStatus.state.holding AND NOT "Unit1.EmNodes".unitStatus.state.held) AND #globalStatus.clock.cycle1000Msec;
   "BA010AZCRSP202.15" := ("BA010AZCRSP201.00" AND "Unit1.ControlNodes".AutoStartEnable AND NOT #instTonTimer[1].Q) OR "Unit1.EmNodes".signalStack.horn OR ("Unit1.EmNodes".unitStatus.mode.production AND "Unit1.EmNodes".unitStatus.specialFunctions.reWrokMode AND ("Unit1.Alarms".unitAlarms.error OR "Unit1.EmNodes".unitStatus.state.complete) AND "Global.Data".general.clock.cycle1000Msec);
END_REGION

REGION Network 22: Q-DAS ReelCut Inspection Data Mapping
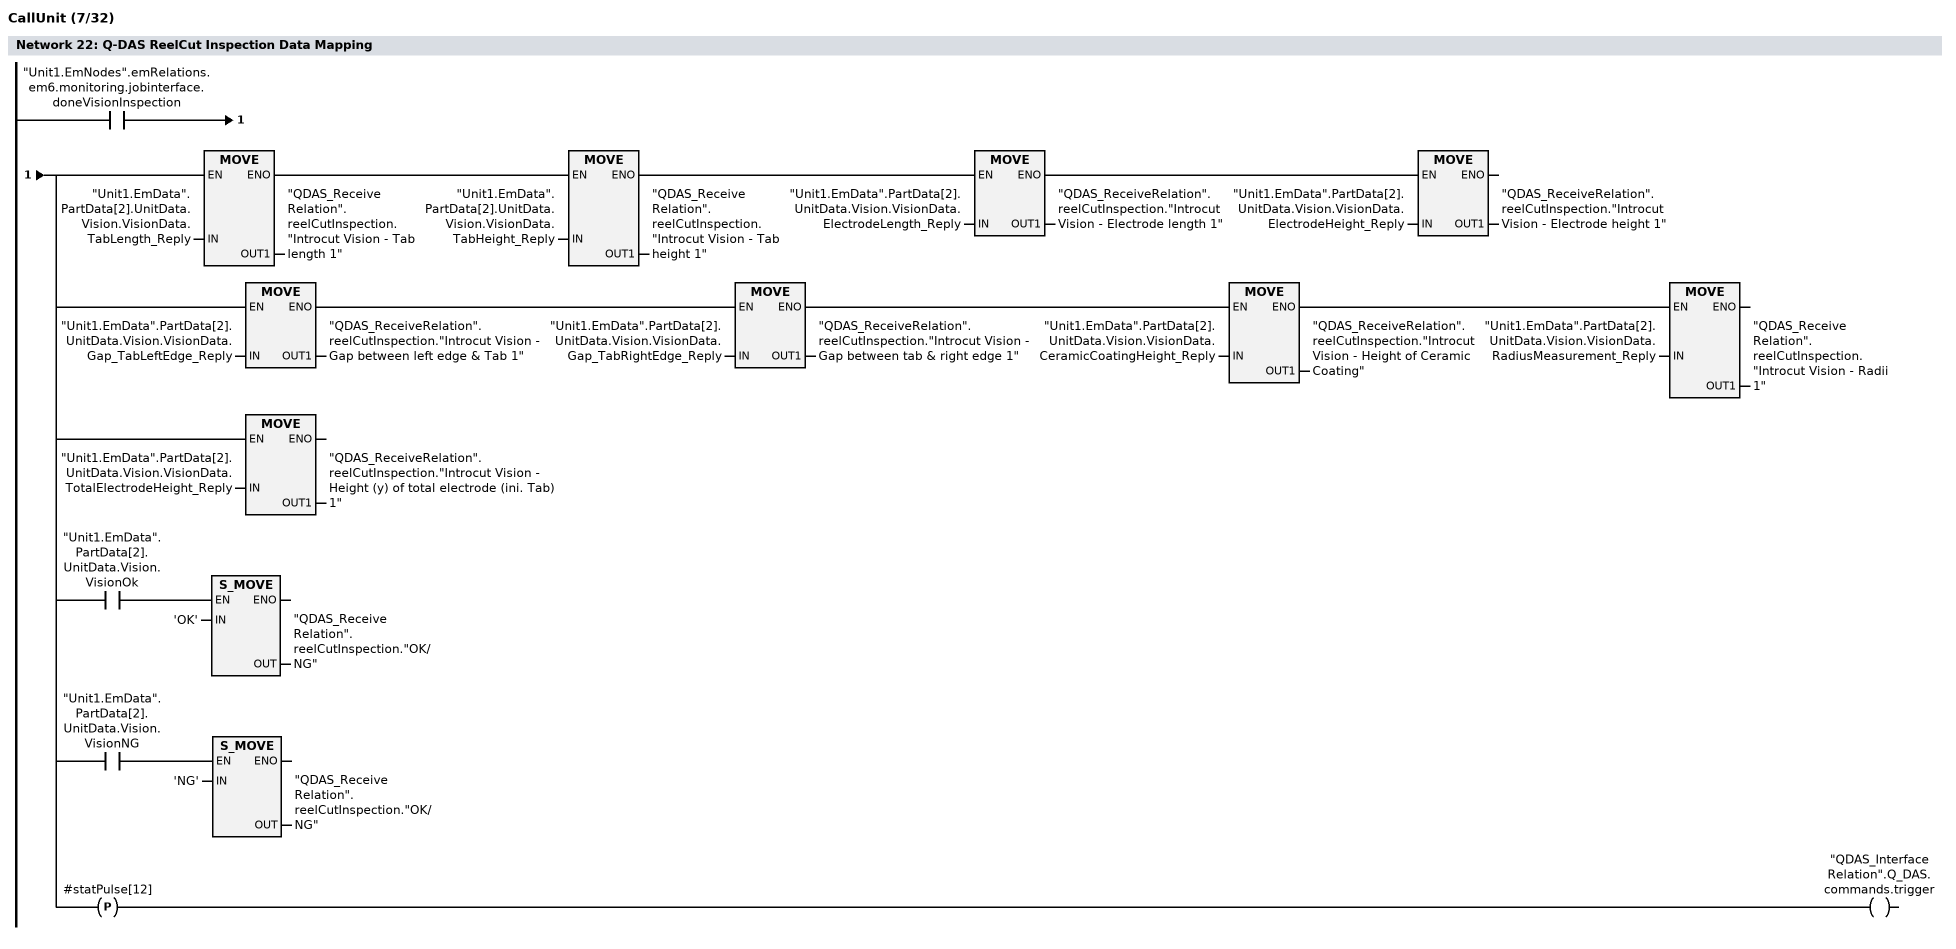
   IF "Unit1.EmNodes".emRelations.em6.monitoring.jobinterface.doneVisionInspection THEN
       "QDAS_ReceiveRelation".reelCutInspection."Introcut Vision - Tab length 1" := "Unit1.EmData".PartData[2].UnitData.Vision.VisionData.TabLength_Reply;
       "QDAS_ReceiveRelation".reelCutInspection."Introcut Vision - Tab height 1" := "Unit1.EmData".PartData[2].UnitData.Vision.VisionData.TabHeight_Reply;
       "QDAS_ReceiveRelation".reelCutInspection."Introcut Vision - Electrode length 1" := "Unit1.EmData".PartData[2].UnitData.Vision.VisionData.ElectrodeLength_Reply;
       "QDAS_ReceiveRelation".reelCutInspection."Introcut Vision - Electrode height 1" := "Unit1.EmData".PartData[2].UnitData.Vision.VisionData.ElectrodeHeight_Reply;
       "QDAS_ReceiveRelation".reelCutInspection."Introcut Vision - Gap between left edge & Tab 1" := "Unit1.EmData".PartData[2].UnitData.Vision.VisionData.Gap_TabLeftEdge_Reply;
       "QDAS_ReceiveRelation".reelCutInspection."Introcut Vision - Gap between tab & right edge 1" := "Unit1.EmData".PartData[2].UnitData.Vision.VisionData.Gap_TabRightEdge_Reply;
       "QDAS_ReceiveRelation".reelCutInspection."Introcut Vision - Height of Ceramic Coating" := "Unit1.EmData".PartData[2].UnitData.Vision.VisionData.CeramicCoatingHeight_Reply;
       "QDAS_ReceiveRelation".reelCutInspection."Introcut Vision - Radii 1" := "Unit1.EmData".PartData[2].UnitData.Vision.VisionData.RadiusMeasurement_Reply;
       "QDAS_ReceiveRelation".reelCutInspection."Introcut Vision - Height (y) of total electrode (ini. Tab) 1" := "Unit1.EmData".PartData[2].UnitData.Vision.VisionData.TotalElectrodeHeight_Reply;
   END_IF;
   IF "Unit1.EmNodes".emRelations.em6.monitoring.jobinterface.doneVisionInspection AND "Unit1.EmData".PartData[2].UnitData.Vision.VisionOk THEN
       "QDAS_ReceiveRelation".reelCutInspection."OK/NG" := 'OK';
   END_IF;
   IF "Unit1.EmNodes".emRelations.em6.monitoring.jobinterface.doneVisionInspection AND "Unit1.EmData".PartData[2].UnitData.Vision.VisionNG THEN
       "QDAS_ReceiveRelation".reelCutInspection."OK/NG" := 'NG';
   END_IF;
   #_w1 := "Unit1.EmNodes".emRelations.em6.monitoring.jobinterface.doneVisionInspection AND NOT #statPulse[12];   // rising edge
   #statPulse[12] := "Unit1.EmNodes".emRelations.em6.monitoring.jobinterface.doneVisionInspection;
   "QDAS_InterfaceRelation".Q_DAS.commands.trigger := #_w1;
END_REGION

REGION Network 23: Remote Control via OPC UA
   // Control the mode state manager remotely via OPC UA
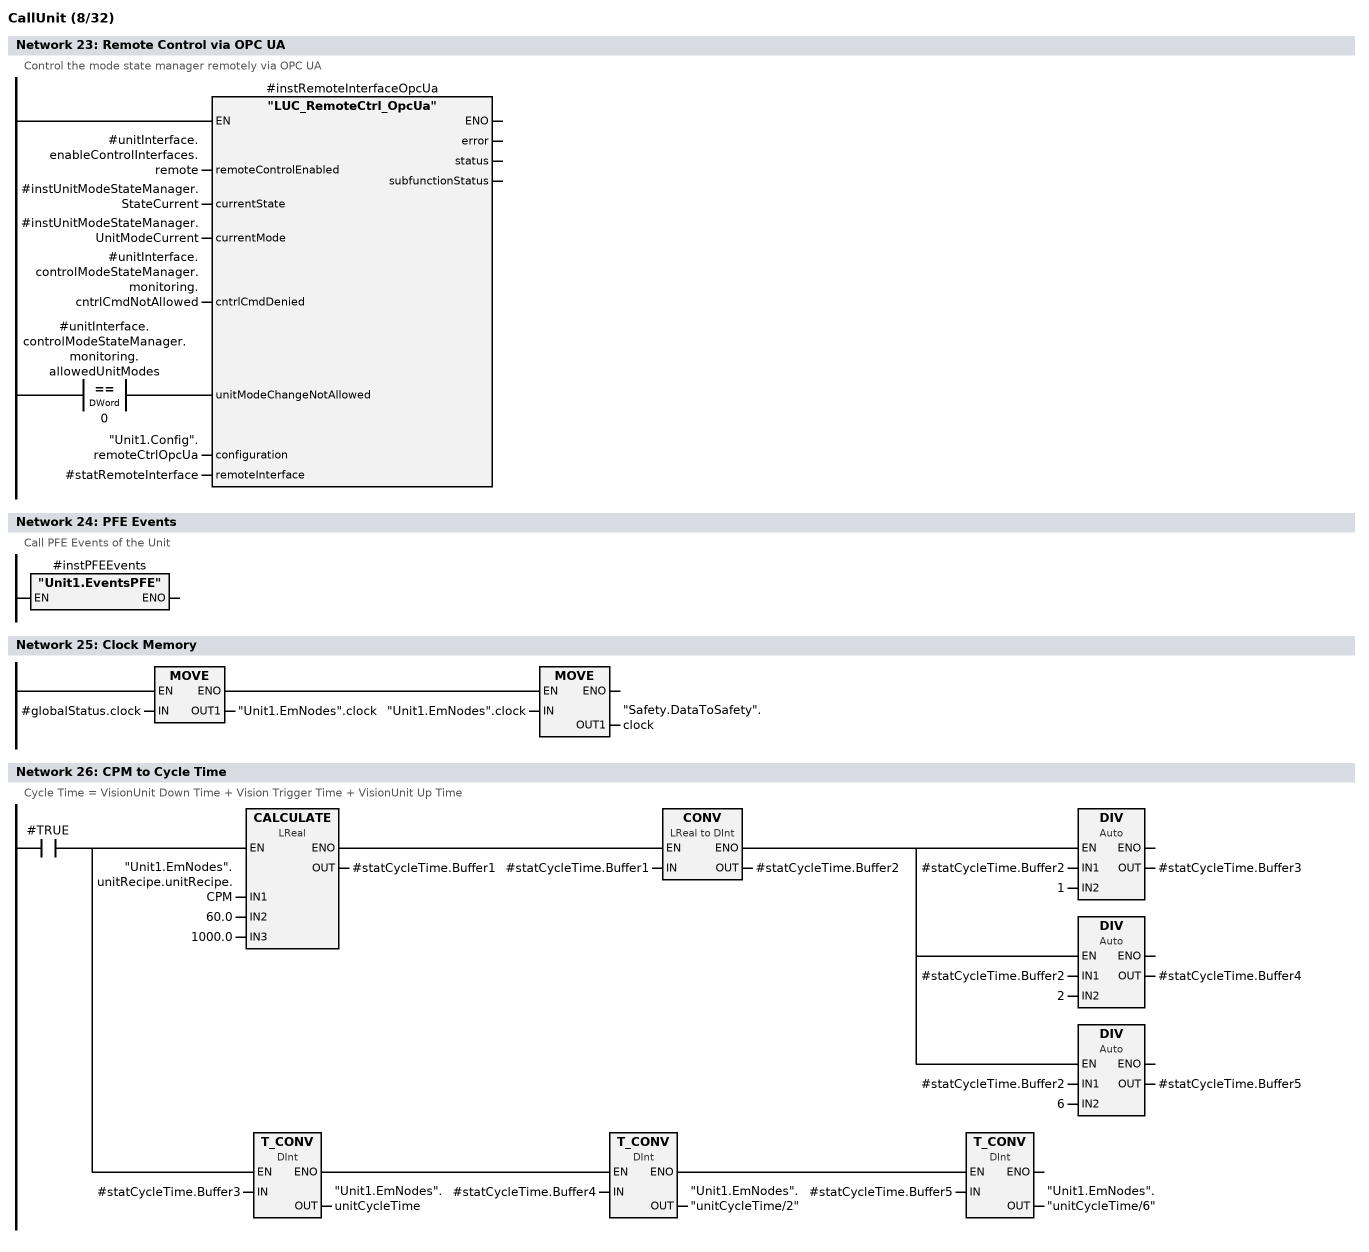
   RUNG wire#powerrail
      #instRemoteInterfaceOpcUa(unitModeChangeNotAllowed := wire#w1, remoteControlEnabled := #unitInterface.enableControlInterfaces.remote, currentState := #instUnitModeStateManager.StateCurrent, currentMode := #instUnitModeStateManager.UnitModeCurrent, cntrlCmdDenied := #unitInterface.controlModeStateManager.monitoring.cntrlCmdNotAllowed, configuration := "Unit1.Config".remoteCtrlOpcUa, remoteInterface := #statRemoteInterface, error =>, status =>, subfunctionStatus =>)
   END_RUNG
   RUNG wire#powerrail
      { S7_Templates := "SrcType := DWord" } EQ_Contact(in1 := #unitInterface.controlModeStateManager.monitoring.allowedUnitModes, in2 := 0)
   END_RUNG wire#w1
   // the same network as SCL:
   #instRemoteInterfaceOpcUa(remoteControlEnabled := #unitInterface.enableControlInterfaces.remote,   // "LUC_RemoteCtrl_OpcUa"
                           currentState := #instUnitModeStateManager.StateCurrent,
                           currentMode := #instUnitModeStateManager.UnitModeCurrent,
                           cntrlCmdDenied := #unitInterface.controlModeStateManager.monitoring.cntrlCmdNotAllowed,
                           unitModeChangeNotAllowed := #unitInterface.controlModeStateManager.monitoring.allowedUnitModes = 0,
                           configuration := "Unit1.Config".remoteCtrlOpcUa,
                           remoteInterface := #statRemoteInterface);
END_REGION

REGION Network 24: PFE Events
   // Call PFE Events of the Unit
   RUNG wire#powerrail
      #instPFEEvents()
   END_RUNG
   // the same network as SCL:
   #instPFEEvents();   // "Unit1.EventsPFE"
END_REGION

REGION Network 25: Clock Memory
   RUNG wire#powerrail
      Move(in := #globalStatus.clock, out1 => "Unit1.EmNodes".clock)
      Move(in := "Unit1.EmNodes".clock, out1 => "Safety.DataToSafety".clock)
   END_RUNG
   // the same network as SCL:
   "Unit1.EmNodes".clock := #globalStatus.clock;
   "Safety.DataToSafety".clock := "Unit1.EmNodes".clock;
END_REGION

REGION Network 26: CPM to Cycle Time
   // Cycle Time = VisionUnit Down Time + Vision Trigger Time + VisionUnit Up Time
   RUNG wire#powerrail
      Contact( #TRUE )
      wire#w1
      { S7_Templates := "SrcType := LReal"; S7_Expression := "(IN2/IN1)*IN3" } Calculate(in1 := "Unit1.EmNodes".unitRecipe.unitRecipe.CPM, in2 := 60.0, in3 := 1000.0, out => #statCycleTime.Buffer1)
      { S7_Templates := "[SrcType := LReal, DestType := DInt]" } Convert(in := #statCycleTime.Buffer1, out => #statCycleTime.Buffer2)
      wire#w2
      Div(in1 := #statCycleTime.Buffer2, in2 := 1, out => #statCycleTime.Buffer3)
   END_RUNG
   RUNG wire#w2
      Div(in1 := #statCycleTime.Buffer2, in2 := 2, out => #statCycleTime.Buffer4)
   END_RUNG
   RUNG wire#w2
      Div(in1 := #statCycleTime.Buffer2, in2 := 6, out => #statCycleTime.Buffer5)
   END_RUNG
   RUNG wire#w1
      { S7_Templates := "[src_type := DInt, dest_type := Time]" } T_CONV(IN := #statCycleTime.Buffer3, OUT => "Unit1.EmNodes".unitCycleTime)
      { S7_Templates := "[src_type := DInt, dest_type := Time]" } T_CONV(IN := #statCycleTime.Buffer4, OUT => "Unit1.EmNodes"."unitCycleTime/2")
      { S7_Templates := "[src_type := DInt, dest_type := Time]" } T_CONV(IN := #statCycleTime.Buffer5, OUT => "Unit1.EmNodes"."unitCycleTime/6")
   END_RUNG
   // the same network as SCL:
   IF #TRUE THEN
       #statCycleTime.Buffer1 := (60.0/"Unit1.EmNodes".unitRecipe.unitRecipe.CPM)*1000.0;
       #statCycleTime.Buffer2 := LREAL_TO_DINT(#statCycleTime.Buffer1);
       #statCycleTime.Buffer3 := #statCycleTime.Buffer2 / 1;
       #statCycleTime.Buffer4 := #statCycleTime.Buffer2 / 2;
       #statCycleTime.Buffer5 := #statCycleTime.Buffer2 / 6;
   END_IF;
   T_CONV(EN := #TRUE, IN := #statCycleTime.Buffer3, OUT => "Unit1.EmNodes".unitCycleTime, ENO => #_w1);
   T_CONV(EN := #_w1, IN := #statCycleTime.Buffer4, OUT => "Unit1.EmNodes"."unitCycleTime/2", ENO => #_w2);
   IF #_w2 THEN T_CONV(IN := #statCycleTime.Buffer5, OUT => "Unit1.EmNodes"."unitCycleTime/6"); END_IF;
END_REGION

REGION Network 27: ******************** Power ********************
END_REGION

REGION Network 28: LED Power
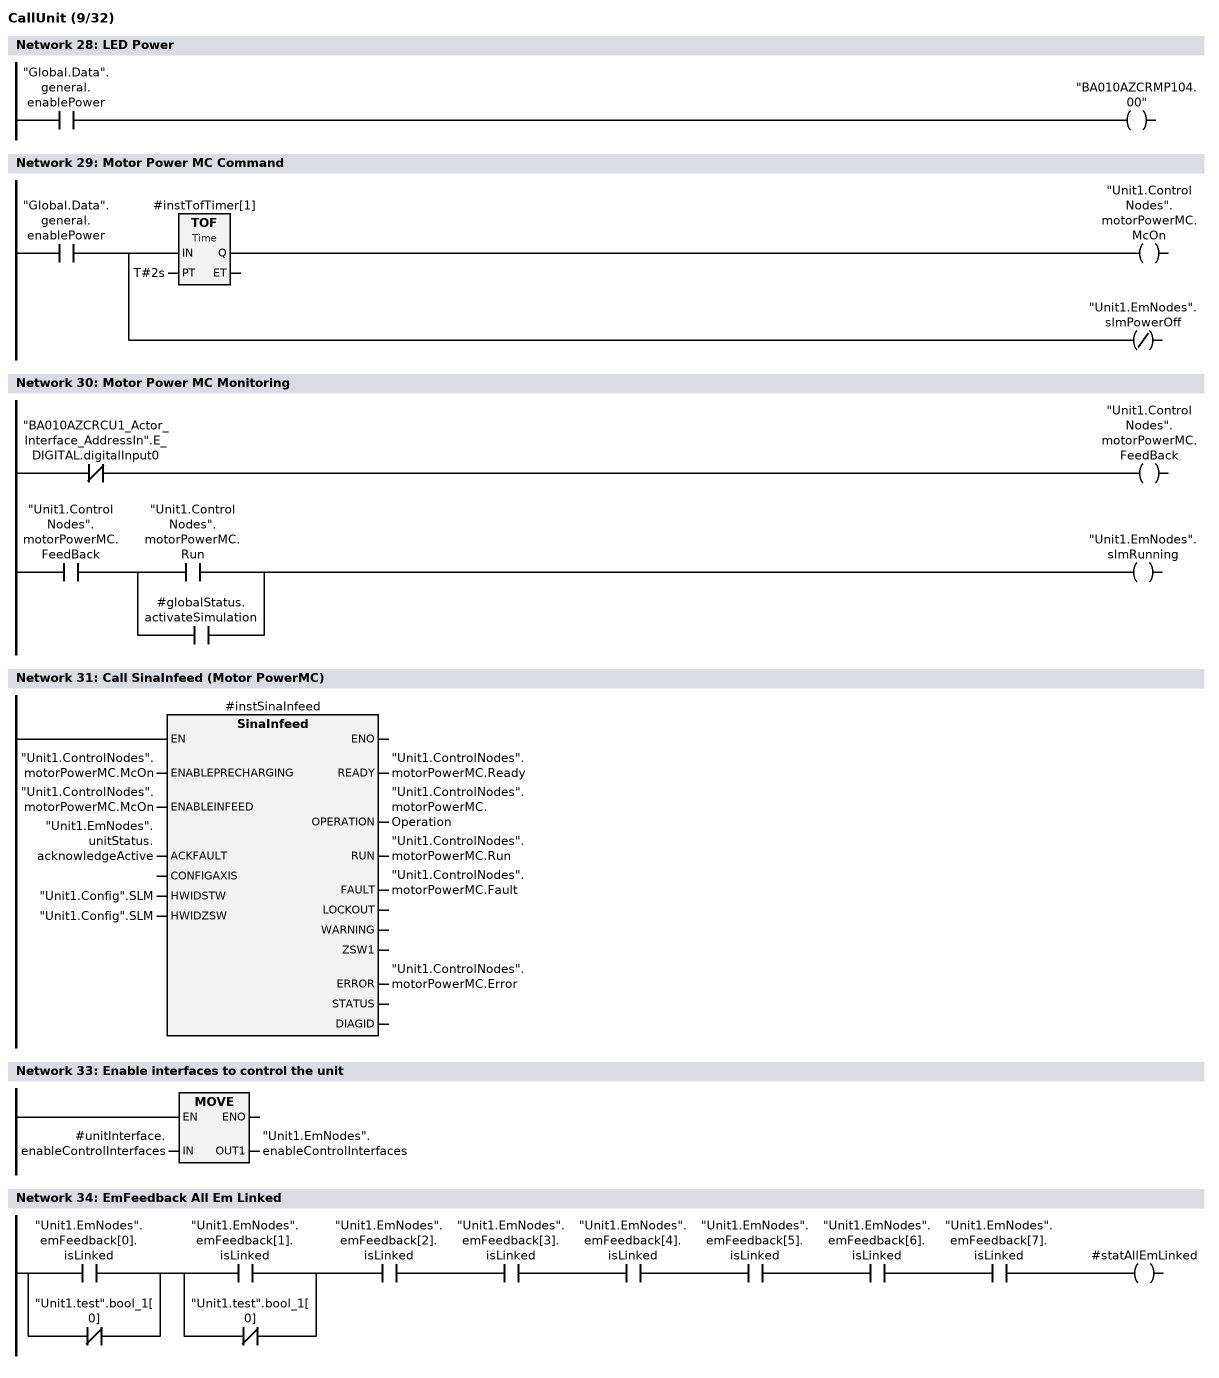
   RUNG wire#powerrail
      Contact( "Global.Data".general.enablePower )
      Coil( "BA010AZCRMP104.00" )
   END_RUNG
   // the same network as SCL:
   "BA010AZCRMP104.00" := "Global.Data".general.enablePower;
END_REGION

REGION Network 29: Motor Power MC Command
   RUNG wire#powerrail
      Contact( "Global.Data".general.enablePower )
      wire#w1
      { S7_Templates := "time_type := Time" } #instTofTimer[1].TOF(pt := T#2s, et =>)
      Coil( "Unit1.ControlNodes".motorPowerMC.McOn )
   END_RUNG
   RUNG wire#w1
      I_Coil( "Unit1.EmNodes".slmPowerOff )
   END_RUNG
   // the same network as SCL:
   #instTofTimer[1].TOF(IN := "Global.Data".general.enablePower, PT := T#2s);
   "Unit1.ControlNodes".motorPowerMC.McOn := #instTofTimer[1].Q;
   "Unit1.EmNodes".slmPowerOff := NOT "Global.Data".general.enablePower;
END_REGION

REGION Network 30: Motor Power MC Monitoring
   RUNG wire#powerrail
      I_Contact( "BA010AZCRCU1_Actor_Interface_AddressIn".E_DIGITAL.digitalInput0 )
      Coil( "Unit1.ControlNodes".motorPowerMC.FeedBack )
   END_RUNG
   RUNG wire#powerrail
      Contact( "Unit1.ControlNodes".motorPowerMC.FeedBack )
      wire#w1
      Contact( "Unit1.ControlNodes".motorPowerMC.Run )
      wire#w2
      Coil( "Unit1.EmNodes".slmRunning )
   END_RUNG
   RUNG wire#w1
      Contact( #globalStatus.activateSimulation )
   END_RUNG wire#w2
   // the same network as SCL:
   "Unit1.ControlNodes".motorPowerMC.FeedBack := NOT "BA010AZCRCU1_Actor_Interface_AddressIn".E_DIGITAL.digitalInput0;
   "Unit1.EmNodes".slmRunning := "Unit1.ControlNodes".motorPowerMC.FeedBack AND ("Unit1.ControlNodes".motorPowerMC.Run OR #globalStatus.activateSimulation);
END_REGION

REGION Network 31: Call SinaInfeed (Motor PowerMC)
   RUNG wire#powerrail
      #instSinaInfeed.SinaInfeed(EnablePrecharging := "Unit1.ControlNodes".motorPowerMC.McOn, EnableInfeed := "Unit1.ControlNodes".motorPowerMC.McOn, AckFault := "Unit1.EmNodes".unitStatus.acknowledgeActive, ConfigAxis :=, HWIDSTW := "Unit1.Config".SLM, HWIDZSW := "Unit1.Config".SLM, Ready => "Unit1.ControlNodes".motorPowerMC.Ready, Operation => "Unit1.ControlNodes".motorPowerMC.Operation, Run => "Unit1.ControlNodes".motorPowerMC.Run, Fault => "Unit1.ControlNodes".motorPowerMC.Fault, Lockout =>, Warning =>, ZSW1 =>, Error => "Unit1.ControlNodes".motorPowerMC.Error, Status =>, DiagID =>)
   END_RUNG
   // the same network as SCL:
   #instSinaInfeed(EnablePrecharging := "Unit1.ControlNodes".motorPowerMC.McOn,   // SinaInfeed
                   EnableInfeed := "Unit1.ControlNodes".motorPowerMC.McOn,
                   AckFault := "Unit1.EmNodes".unitStatus.acknowledgeActive,
                   HWIDSTW := "Unit1.Config".SLM,
                   HWIDZSW := "Unit1.Config".SLM,
                   Ready => "Unit1.ControlNodes".motorPowerMC.Ready,
                   Operation => "Unit1.ControlNodes".motorPowerMC.Operation,
                   Run => "Unit1.ControlNodes".motorPowerMC.Run,
                   Fault => "Unit1.ControlNodes".motorPowerMC.Fault,
                   Error => "Unit1.ControlNodes".motorPowerMC.Error);
END_REGION

REGION Network 32: ******************** Local Operation Box ********************
END_REGION

REGION Network 33: Enable interfaces to control the unit
   RUNG wire#powerrail
      Move(in := #unitInterface.enableControlInterfaces, out1 => "Unit1.EmNodes".enableControlInterfaces)
   END_RUNG
   // the same network as SCL:
   "Unit1.EmNodes".enableControlInterfaces := #unitInterface.enableControlInterfaces;
END_REGION

REGION Network 34: EmFeedback All Em Linked
   RUNG wire#powerrail
      Contact( "Unit1.EmNodes".emFeedback[0].isLinked )
      wire#w1
      Contact( "Unit1.EmNodes".emFeedback[1].isLinked )
      wire#w2
      Contact( "Unit1.EmNodes".emFeedback[2].isLinked )
      Contact( "Unit1.EmNodes".emFeedback[3].isLinked )
      Contact( "Unit1.EmNodes".emFeedback[4].isLinked )
      Contact( "Unit1.EmNodes".emFeedback[5].isLinked )
      Contact( "Unit1.EmNodes".emFeedback[6].isLinked )
      Contact( "Unit1.EmNodes".emFeedback[7].isLinked )
      Coil( #statAllEmLinked )
   END_RUNG
   RUNG wire#powerrail
      I_Contact( "Unit1.test".bool_1[0] )
   END_RUNG wire#w1
   RUNG wire#w1
      I_Contact( "Unit1.test".bool_1[0] )
   END_RUNG wire#w2
   // the same network as SCL:
   #statAllEmLinked := ("Unit1.EmNodes".emFeedback[0].isLinked OR NOT "Unit1.test".bool_1[0]) AND ("Unit1.EmNodes".emFeedback[1].isLinked OR NOT "Unit1.test".bool_1[0]) AND "Unit1.EmNodes".emFeedback[2].isLinked AND "Unit1.EmNodes".emFeedback[3].isLinked AND "Unit1.EmNodes".emFeedback[4].isLinked AND "Unit1.EmNodes".emFeedback[5].isLinked AND "Unit1.EmNodes".emFeedback[6].isLinked AND "Unit1.EmNodes".emFeedback[7].isLinked;
END_REGION

REGION Network 35: EM Enable Check
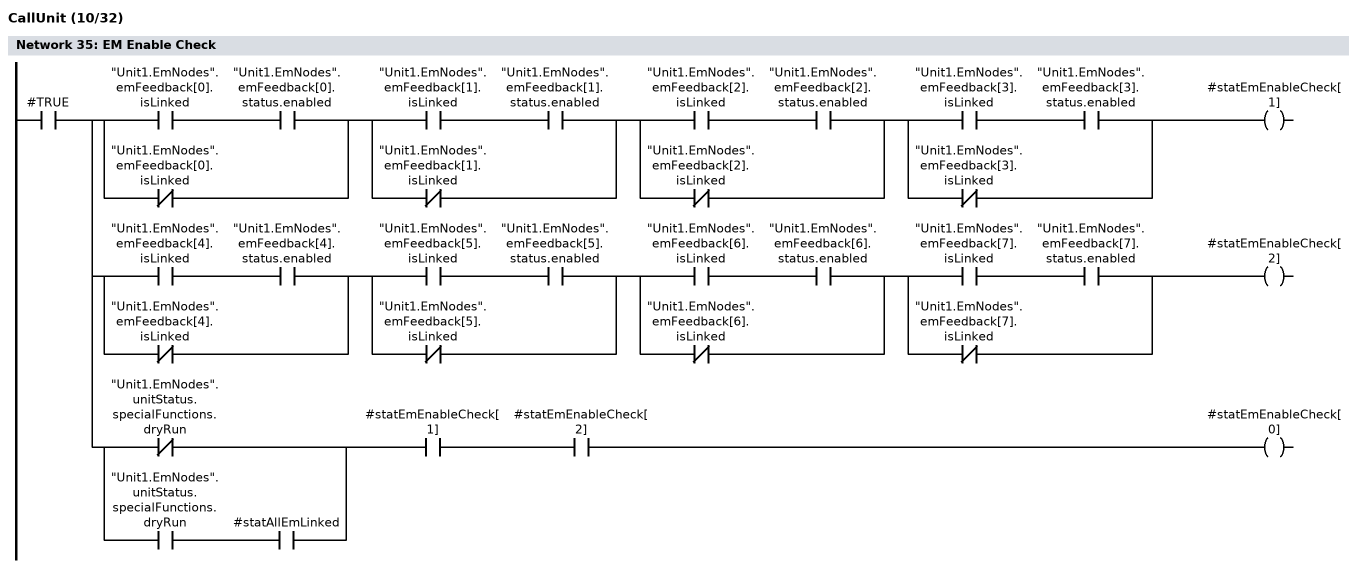
   RUNG wire#powerrail
      Contact( #TRUE )
      wire#w1
      Contact( "Unit1.EmNodes".emFeedback[0].isLinked )
      Contact( "Unit1.EmNodes".emFeedback[0].status.enabled )
      wire#w2
      Contact( "Unit1.EmNodes".emFeedback[1].isLinked )
      Contact( "Unit1.EmNodes".emFeedback[1].status.enabled )
      wire#w3
      Contact( "Unit1.EmNodes".emFeedback[2].isLinked )
      Contact( "Unit1.EmNodes".emFeedback[2].status.enabled )
      wire#w4
      Contact( "Unit1.EmNodes".emFeedback[3].isLinked )
      Contact( "Unit1.EmNodes".emFeedback[3].status.enabled )
      wire#w5
      Coil( #statEmEnableCheck[1] )
   END_RUNG
   RUNG wire#w1
      I_Contact( "Unit1.EmNodes".emFeedback[0].isLinked )
   END_RUNG wire#w2
   RUNG wire#w2
      I_Contact( "Unit1.EmNodes".emFeedback[1].isLinked )
   END_RUNG wire#w3
   RUNG wire#w3
      I_Contact( "Unit1.EmNodes".emFeedback[2].isLinked )
   END_RUNG wire#w4
   RUNG wire#w4
      I_Contact( "Unit1.EmNodes".emFeedback[3].isLinked )
   END_RUNG wire#w5
   RUNG wire#w1
      Contact( "Unit1.EmNodes".emFeedback[4].isLinked )
      Contact( "Unit1.EmNodes".emFeedback[4].status.enabled )
      wire#w6
      Contact( "Unit1.EmNodes".emFeedback[5].isLinked )
      Contact( "Unit1.EmNodes".emFeedback[5].status.enabled )
      wire#w7
      Contact( "Unit1.EmNodes".emFeedback[6].isLinked )
      Contact( "Unit1.EmNodes".emFeedback[6].status.enabled )
      wire#w8
      Contact( "Unit1.EmNodes".emFeedback[7].isLinked )
      Contact( "Unit1.EmNodes".emFeedback[7].status.enabled )
      wire#w9
      Coil( #statEmEnableCheck[2] )
   END_RUNG
   RUNG wire#w1
      I_Contact( "Unit1.EmNodes".emFeedback[4].isLinked )
   END_RUNG wire#w6
   RUNG wire#w6
      I_Contact( "Unit1.EmNodes".emFeedback[5].isLinked )
   END_RUNG wire#w7
   RUNG wire#w7
      I_Contact( "Unit1.EmNodes".emFeedback[6].isLinked )
   END_RUNG wire#w8
   RUNG wire#w8
      I_Contact( "Unit1.EmNodes".emFeedback[7].isLinked )
   END_RUNG wire#w9
   RUNG wire#w1
      I_Contact( "Unit1.EmNodes".unitStatus.specialFunctions.dryRun )
      wire#w10
      Contact( #statEmEnableCheck[1] )
      Contact( #statEmEnableCheck[2] )
      Coil( #statEmEnableCheck[0] )
   END_RUNG
   RUNG wire#w1
      Contact( "Unit1.EmNodes".unitStatus.specialFunctions.dryRun )
      Contact( #statAllEmLinked )
   END_RUNG wire#w10
   // the same network as SCL:
   #statEmEnableCheck[1] := #TRUE AND (("Unit1.EmNodes".emFeedback[0].isLinked AND "Unit1.EmNodes".emFeedback[0].status.enabled) OR NOT "Unit1.EmNodes".emFeedback[0].isLinked) AND (("Unit1.EmNodes".emFeedback[1].isLinked AND "Unit1.EmNodes".emFeedback[1].status.enabled) OR NOT "Unit1.EmNodes".emFeedback[1].isLinked) AND (("Unit1.EmNodes".emFeedback[2].isLinked AND "Unit1.EmNodes".emFeedback[2].status.enabled) OR NOT "Unit1.EmNodes".emFeedback[2].isLinked) AND (("Unit1.EmNodes".emFeedback[3].isLinked AND "Unit1.EmNodes".emFeedback[3].status.enabled) OR NOT "Unit1.EmNodes".emFeedback[3].isLinked);
   #statEmEnableCheck[2] := #TRUE AND (("Unit1.EmNodes".emFeedback[4].isLinked AND "Unit1.EmNodes".emFeedback[4].status.enabled) OR NOT "Unit1.EmNodes".emFeedback[4].isLinked) AND (("Unit1.EmNodes".emFeedback[5].isLinked AND "Unit1.EmNodes".emFeedback[5].status.enabled) OR NOT "Unit1.EmNodes".emFeedback[5].isLinked) AND (("Unit1.EmNodes".emFeedback[6].isLinked AND "Unit1.EmNodes".emFeedback[6].status.enabled) OR NOT "Unit1.EmNodes".emFeedback[6].isLinked) AND (("Unit1.EmNodes".emFeedback[7].isLinked AND "Unit1.EmNodes".emFeedback[7].status.enabled) OR NOT "Unit1.EmNodes".emFeedback[7].isLinked);
   #statEmEnableCheck[0] := #TRUE AND (NOT "Unit1.EmNodes".unitStatus.specialFunctions.dryRun OR ("Unit1.EmNodes".unitStatus.specialFunctions.dryRun AND #statAllEmLinked)) AND #statEmEnableCheck[1] AND #statEmEnableCheck[2];
END_REGION

REGION Network 36: Unit State Commands Starting Enable
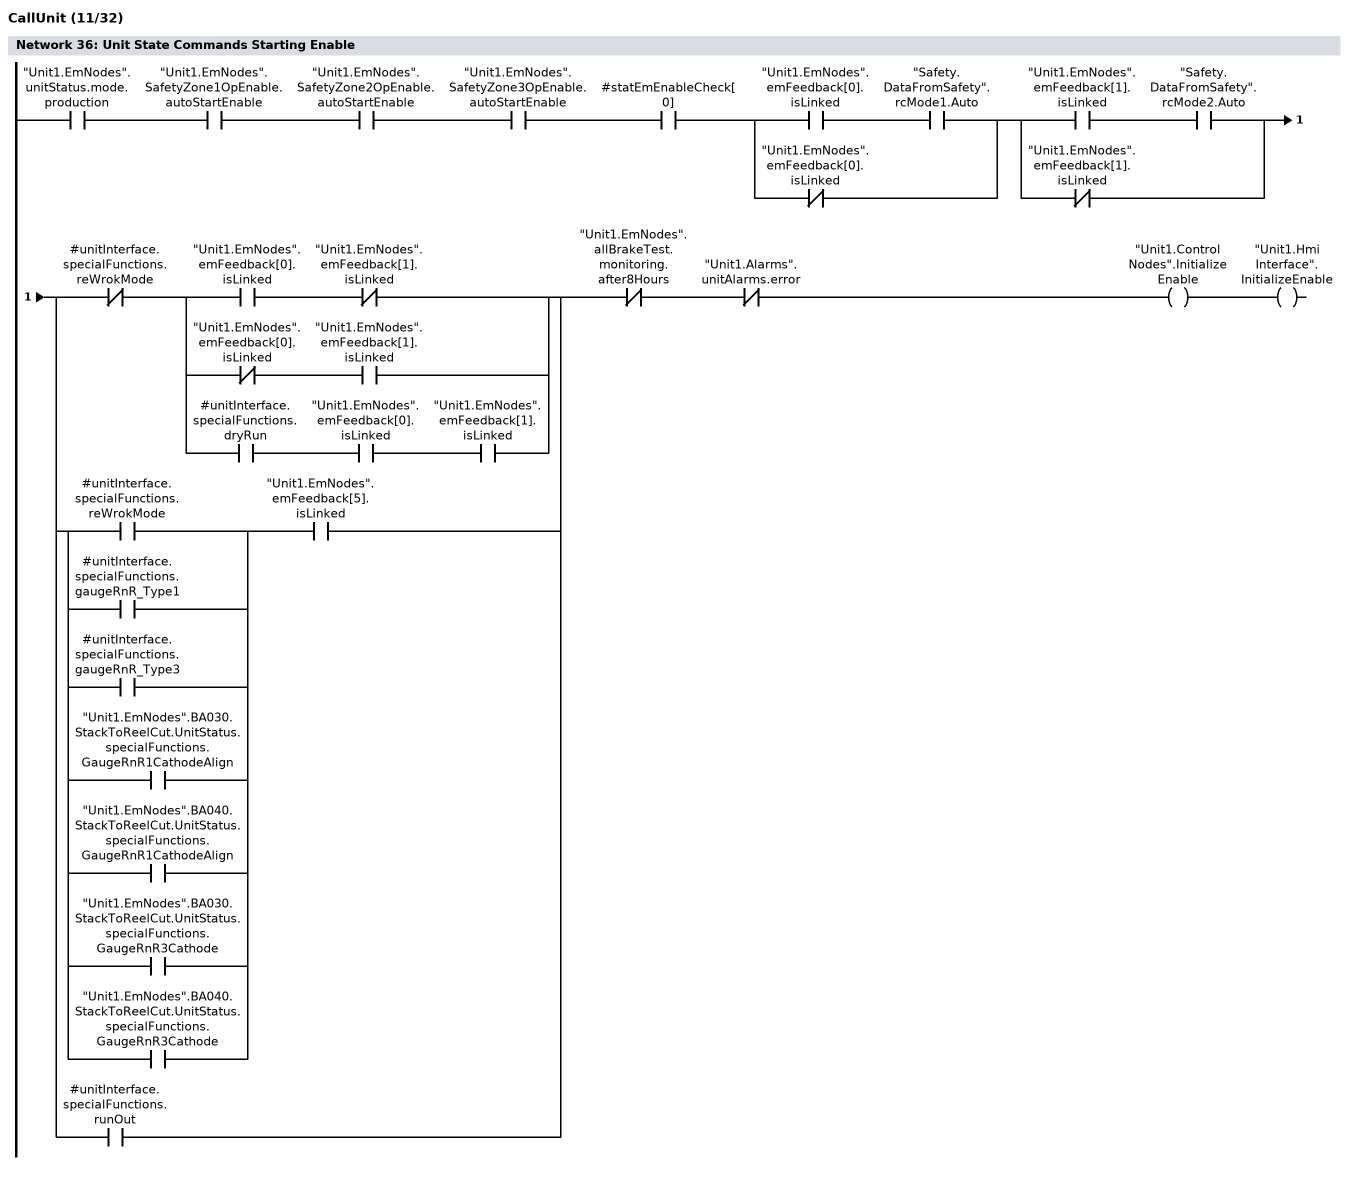
   RUNG wire#powerrail
      Contact( "Unit1.EmNodes".unitStatus.mode.production )
      Contact( "Unit1.EmNodes".SafetyZone1OpEnable.autoStartEnable )
      Contact( "Unit1.EmNodes".SafetyZone2OpEnable.autoStartEnable )
      Contact( "Unit1.EmNodes".SafetyZone3OpEnable.autoStartEnable )
      Contact( #statEmEnableCheck[0] )
      wire#w1
      Contact( "Unit1.EmNodes".emFeedback[0].isLinked )
      Contact( "Safety.DataFromSafety".rcMode1.Auto )
      wire#w2
      Contact( "Unit1.EmNodes".emFeedback[1].isLinked )
      Contact( "Safety.DataFromSafety".rcMode2.Auto )
      wire#w3
      I_Contact( #unitInterface.specialFunctions.reWrokMode )
      wire#w4
      Contact( "Unit1.EmNodes".emFeedback[0].isLinked )
      I_Contact( "Unit1.EmNodes".emFeedback[1].isLinked )
      wire#w5
      I_Contact( "Unit1.EmNodes".allBrakeTest.monitoring.after8Hours )
      I_Contact( "Unit1.Alarms".unitAlarms.error )
      Coil( "Unit1.ControlNodes".InitializeEnable )
      Coil( "Unit1.HmiInterface".InitializeEnable )
   END_RUNG
   RUNG wire#w1
      I_Contact( "Unit1.EmNodes".emFeedback[0].isLinked )
   END_RUNG wire#w2
   RUNG wire#w2
      I_Contact( "Unit1.EmNodes".emFeedback[1].isLinked )
   END_RUNG wire#w3
   RUNG wire#w4
      I_Contact( "Unit1.EmNodes".emFeedback[0].isLinked )
      Contact( "Unit1.EmNodes".emFeedback[1].isLinked )
   END_RUNG wire#w5
   RUNG wire#w4
      Contact( #unitInterface.specialFunctions.dryRun )
      Contact( "Unit1.EmNodes".emFeedback[0].isLinked )
      Contact( "Unit1.EmNodes".emFeedback[1].isLinked )
   END_RUNG wire#w5
   RUNG wire#w3
      Contact( #unitInterface.specialFunctions.reWrokMode )
      wire#w6
      Contact( "Unit1.EmNodes".emFeedback[5].isLinked )
   END_RUNG wire#w5
   RUNG wire#w3
      Contact( #unitInterface.specialFunctions.gaugeRnR_Type1 )
   END_RUNG wire#w6
   RUNG wire#w3
      Contact( #unitInterface.specialFunctions.gaugeRnR_Type3 )
   END_RUNG wire#w6
   RUNG wire#w3
      Contact( "Unit1.EmNodes".BA030.StackToReelCut.UnitStatus.specialFunctions.GaugeRnR1CathodeAlign )
   END_RUNG wire#w6
   RUNG wire#w3
      Contact( "Unit1.EmNodes".BA040.StackToReelCut.UnitStatus.specialFunctions.GaugeRnR1CathodeAlign )
   END_RUNG wire#w6
   RUNG wire#w3
      Contact( "Unit1.EmNodes".BA030.StackToReelCut.UnitStatus.specialFunctions.GaugeRnR3Cathode )
   END_RUNG wire#w6
   RUNG wire#w3
      Contact( "Unit1.EmNodes".BA040.StackToReelCut.UnitStatus.specialFunctions.GaugeRnR3Cathode )
   END_RUNG wire#w6
   RUNG wire#w3
      Contact( #unitInterface.specialFunctions.runOut )
   END_RUNG wire#w5
   // the same network as SCL:
   "Unit1.ControlNodes".InitializeEnable := "Unit1.EmNodes".unitStatus.mode.production AND "Unit1.EmNodes".SafetyZone1OpEnable.autoStartEnable AND "Unit1.EmNodes".SafetyZone2OpEnable.autoStartEnable AND "Unit1.EmNodes".SafetyZone3OpEnable.autoStartEnable AND #statEmEnableCheck[0] AND (("Unit1.EmNodes".emFeedback[0].isLinked AND "Safety.DataFromSafety".rcMode1.Auto) OR NOT "Unit1.EmNodes".emFeedback[0].isLinked) AND (("Unit1.EmNodes".emFeedback[1].isLinked AND "Safety.DataFromSafety".rcMode2.Auto) OR NOT "Unit1.EmNodes".emFeedback[1].isLinked) AND ((NOT #unitInterface.specialFunctions.reWrokMode AND (("Unit1.EmNodes".emFeedback[0].isLinked AND NOT "Unit1.EmNodes".emFeedback[1].isLinked) OR (NOT "Unit1.EmNodes".emFeedback[0].isLinked AND "Unit1.EmNodes".emFeedback[1].isLinked) OR (#unitInterface.specialFunctions.dryRun AND "Unit1.EmNodes".emFeedback[0].isLinked AND "Unit1.EmNodes".emFeedback[1].isLinked))) OR ((#unitInterface.specialFunctions.reWrokMode OR #unitInterface.specialFunctions.gaugeRnR_Type1 OR #unitInterface.specialFunctions.gaugeRnR_Type3 OR "Unit1.EmNodes".BA030.StackToReelCut.UnitStatus.specialFunctions.GaugeRnR1CathodeAlign OR "Unit1.EmNodes".BA040.StackToReelCut.UnitStatus.specialFunctions.GaugeRnR1CathodeAlign OR "Unit1.EmNodes".BA030.StackToReelCut.UnitStatus.specialFunctions.GaugeRnR3Cathode OR "Unit1.EmNodes".BA040.StackToReelCut.UnitStatus.specialFunctions.GaugeRnR3Cathode) AND "Unit1.EmNodes".emFeedback[5].isLinked) OR #unitInterface.specialFunctions.runOut) AND NOT "Unit1.EmNodes".allBrakeTest.monitoring.after8Hours AND NOT "Unit1.Alarms".unitAlarms.error;
   "Unit1.HmiInterface".InitializeEnable := "Unit1.ControlNodes".InitializeEnable;
END_REGION

REGION Network 37: EM initialized + Homed Check
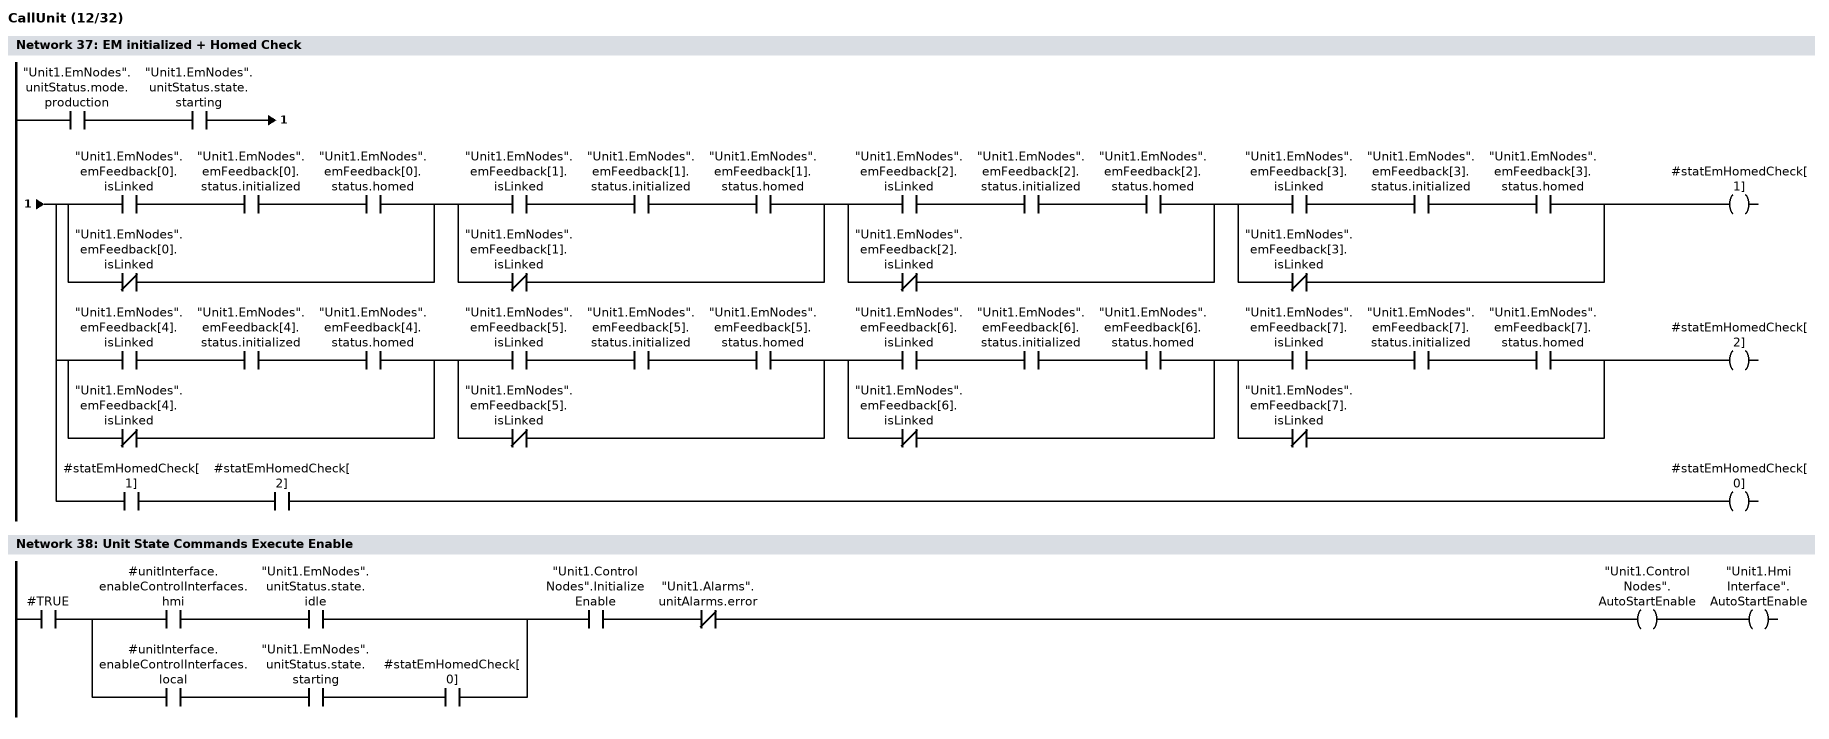
   RUNG wire#powerrail
      Contact( "Unit1.EmNodes".unitStatus.mode.production )
      Contact( "Unit1.EmNodes".unitStatus.state.starting )
      wire#w1
      Contact( "Unit1.EmNodes".emFeedback[0].isLinked )
      Contact( "Unit1.EmNodes".emFeedback[0].status.initialized )
      Contact( "Unit1.EmNodes".emFeedback[0].status.homed )
      wire#w2
      Contact( "Unit1.EmNodes".emFeedback[1].isLinked )
      Contact( "Unit1.EmNodes".emFeedback[1].status.initialized )
      Contact( "Unit1.EmNodes".emFeedback[1].status.homed )
      wire#w3
      Contact( "Unit1.EmNodes".emFeedback[2].isLinked )
      Contact( "Unit1.EmNodes".emFeedback[2].status.initialized )
      Contact( "Unit1.EmNodes".emFeedback[2].status.homed )
      wire#w4
      Contact( "Unit1.EmNodes".emFeedback[3].isLinked )
      Contact( "Unit1.EmNodes".emFeedback[3].status.initialized )
      Contact( "Unit1.EmNodes".emFeedback[3].status.homed )
      wire#w5
      Coil( #statEmHomedCheck[1] )
   END_RUNG
   RUNG wire#w1
      I_Contact( "Unit1.EmNodes".emFeedback[0].isLinked )
   END_RUNG wire#w2
   RUNG wire#w2
      I_Contact( "Unit1.EmNodes".emFeedback[1].isLinked )
   END_RUNG wire#w3
   RUNG wire#w3
      I_Contact( "Unit1.EmNodes".emFeedback[2].isLinked )
   END_RUNG wire#w4
   RUNG wire#w4
      I_Contact( "Unit1.EmNodes".emFeedback[3].isLinked )
   END_RUNG wire#w5
   RUNG wire#w1
      Contact( "Unit1.EmNodes".emFeedback[4].isLinked )
      Contact( "Unit1.EmNodes".emFeedback[4].status.initialized )
      Contact( "Unit1.EmNodes".emFeedback[4].status.homed )
      wire#w6
      Contact( "Unit1.EmNodes".emFeedback[5].isLinked )
      Contact( "Unit1.EmNodes".emFeedback[5].status.initialized )
      Contact( "Unit1.EmNodes".emFeedback[5].status.homed )
      wire#w7
      Contact( "Unit1.EmNodes".emFeedback[6].isLinked )
      Contact( "Unit1.EmNodes".emFeedback[6].status.initialized )
      Contact( "Unit1.EmNodes".emFeedback[6].status.homed )
      wire#w8
      Contact( "Unit1.EmNodes".emFeedback[7].isLinked )
      Contact( "Unit1.EmNodes".emFeedback[7].status.initialized )
      Contact( "Unit1.EmNodes".emFeedback[7].status.homed )
      wire#w9
      Coil( #statEmHomedCheck[2] )
   END_RUNG
   RUNG wire#w1
      I_Contact( "Unit1.EmNodes".emFeedback[4].isLinked )
   END_RUNG wire#w6
   RUNG wire#w6
      I_Contact( "Unit1.EmNodes".emFeedback[5].isLinked )
   END_RUNG wire#w7
   RUNG wire#w7
      I_Contact( "Unit1.EmNodes".emFeedback[6].isLinked )
   END_RUNG wire#w8
   RUNG wire#w8
      I_Contact( "Unit1.EmNodes".emFeedback[7].isLinked )
   END_RUNG wire#w9
   RUNG wire#w1
      Contact( #statEmHomedCheck[1] )
      Contact( #statEmHomedCheck[2] )
      Coil( #statEmHomedCheck[0] )
   END_RUNG
   // the same network as SCL:
   #_w1 := "Unit1.EmNodes".unitStatus.mode.production AND "Unit1.EmNodes".unitStatus.state.starting;
   #statEmHomedCheck[1] := #_w1 AND (("Unit1.EmNodes".emFeedback[0].isLinked AND "Unit1.EmNodes".emFeedback[0].status.initialized AND "Unit1.EmNodes".emFeedback[0].status.homed) OR NOT "Unit1.EmNodes".emFeedback[0].isLinked) AND (("Unit1.EmNodes".emFeedback[1].isLinked AND "Unit1.EmNodes".emFeedback[1].status.initialized AND "Unit1.EmNodes".emFeedback[1].status.homed) OR NOT "Unit1.EmNodes".emFeedback[1].isLinked) AND (("Unit1.EmNodes".emFeedback[2].isLinked AND "Unit1.EmNodes".emFeedback[2].status.initialized AND "Unit1.EmNodes".emFeedback[2].status.homed) OR NOT "Unit1.EmNodes".emFeedback[2].isLinked) AND (("Unit1.EmNodes".emFeedback[3].isLinked AND "Unit1.EmNodes".emFeedback[3].status.initialized AND "Unit1.EmNodes".emFeedback[3].status.homed) OR NOT "Unit1.EmNodes".emFeedback[3].isLinked);
   #statEmHomedCheck[2] := #_w1 AND (("Unit1.EmNodes".emFeedback[4].isLinked AND "Unit1.EmNodes".emFeedback[4].status.initialized AND "Unit1.EmNodes".emFeedback[4].status.homed) OR NOT "Unit1.EmNodes".emFeedback[4].isLinked) AND (("Unit1.EmNodes".emFeedback[5].isLinked AND "Unit1.EmNodes".emFeedback[5].status.initialized AND "Unit1.EmNodes".emFeedback[5].status.homed) OR NOT "Unit1.EmNodes".emFeedback[5].isLinked) AND (("Unit1.EmNodes".emFeedback[6].isLinked AND "Unit1.EmNodes".emFeedback[6].status.initialized AND "Unit1.EmNodes".emFeedback[6].status.homed) OR NOT "Unit1.EmNodes".emFeedback[6].isLinked) AND (("Unit1.EmNodes".emFeedback[7].isLinked AND "Unit1.EmNodes".emFeedback[7].status.initialized AND "Unit1.EmNodes".emFeedback[7].status.homed) OR NOT "Unit1.EmNodes".emFeedback[7].isLinked);
   #statEmHomedCheck[0] := #_w1 AND #statEmHomedCheck[1] AND #statEmHomedCheck[2];
END_REGION

REGION Network 38: Unit State Commands Execute Enable
   RUNG wire#powerrail
      Contact( #TRUE )
      wire#w1
      Contact( #unitInterface.enableControlInterfaces.hmi )
      Contact( "Unit1.EmNodes".unitStatus.state.idle )
      wire#w2
      Contact( "Unit1.ControlNodes".InitializeEnable )
      I_Contact( "Unit1.Alarms".unitAlarms.error )
      Coil( "Unit1.ControlNodes".AutoStartEnable )
      Coil( "Unit1.HmiInterface".AutoStartEnable )
   END_RUNG
   RUNG wire#w1
      Contact( #unitInterface.enableControlInterfaces.local )
      Contact( "Unit1.EmNodes".unitStatus.state.starting )
      Contact( #statEmHomedCheck[0] )
   END_RUNG wire#w2
   // the same network as SCL:
   "Unit1.ControlNodes".AutoStartEnable := #TRUE AND ((#unitInterface.enableControlInterfaces.hmi AND "Unit1.EmNodes".unitStatus.state.idle) OR (#unitInterface.enableControlInterfaces.local AND "Unit1.EmNodes".unitStatus.state.starting AND #statEmHomedCheck[0])) AND "Unit1.ControlNodes".InitializeEnable AND NOT "Unit1.Alarms".unitAlarms.error;
   "Unit1.HmiInterface".AutoStartEnable := "Unit1.ControlNodes".AutoStartEnable;
END_REGION

REGION Network 39: Main Op Local Control
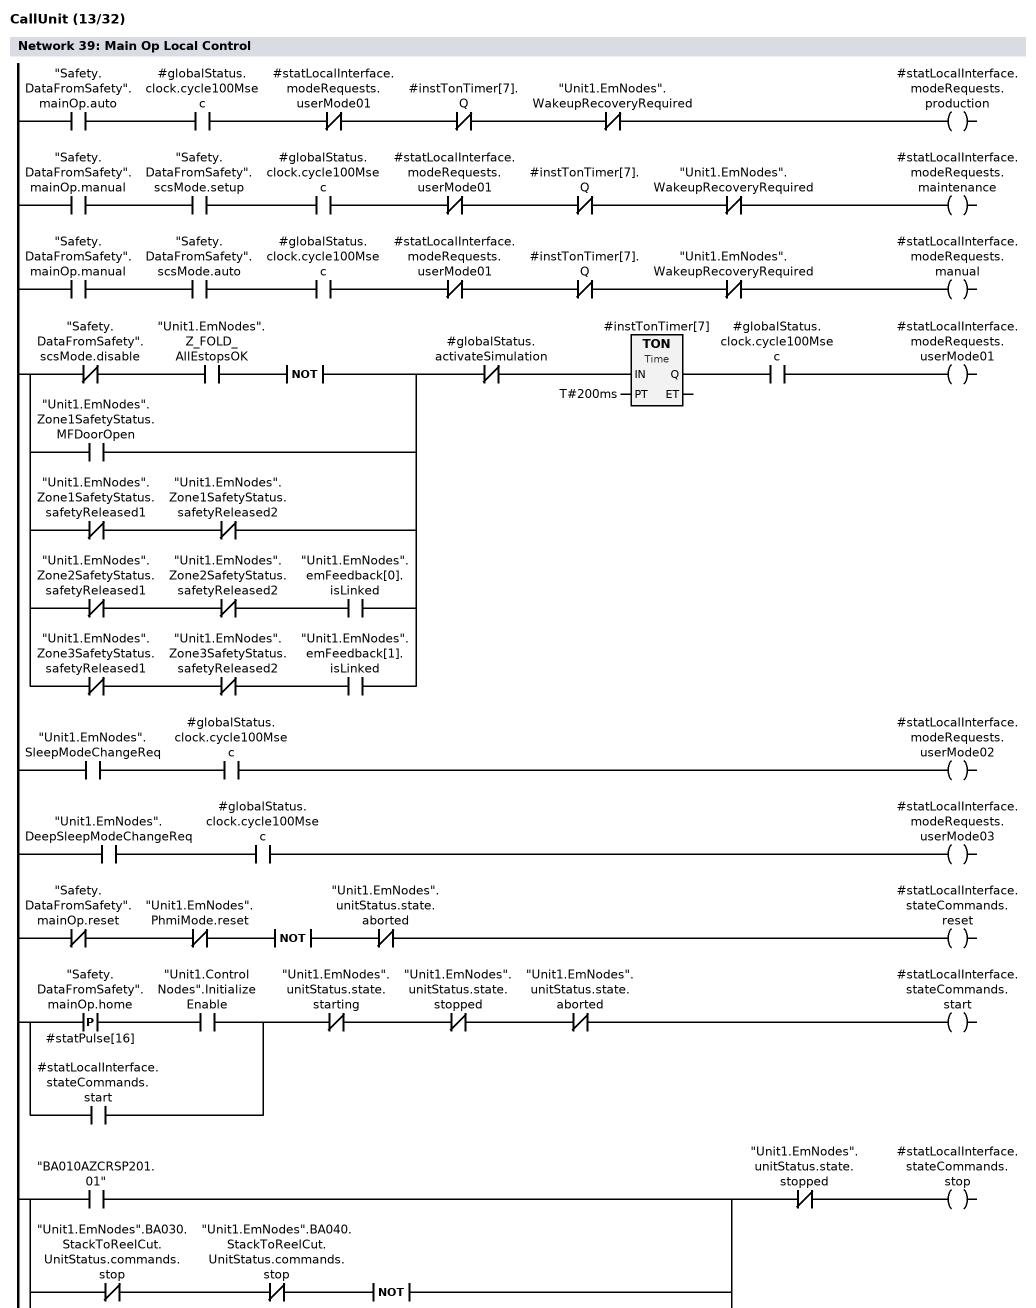
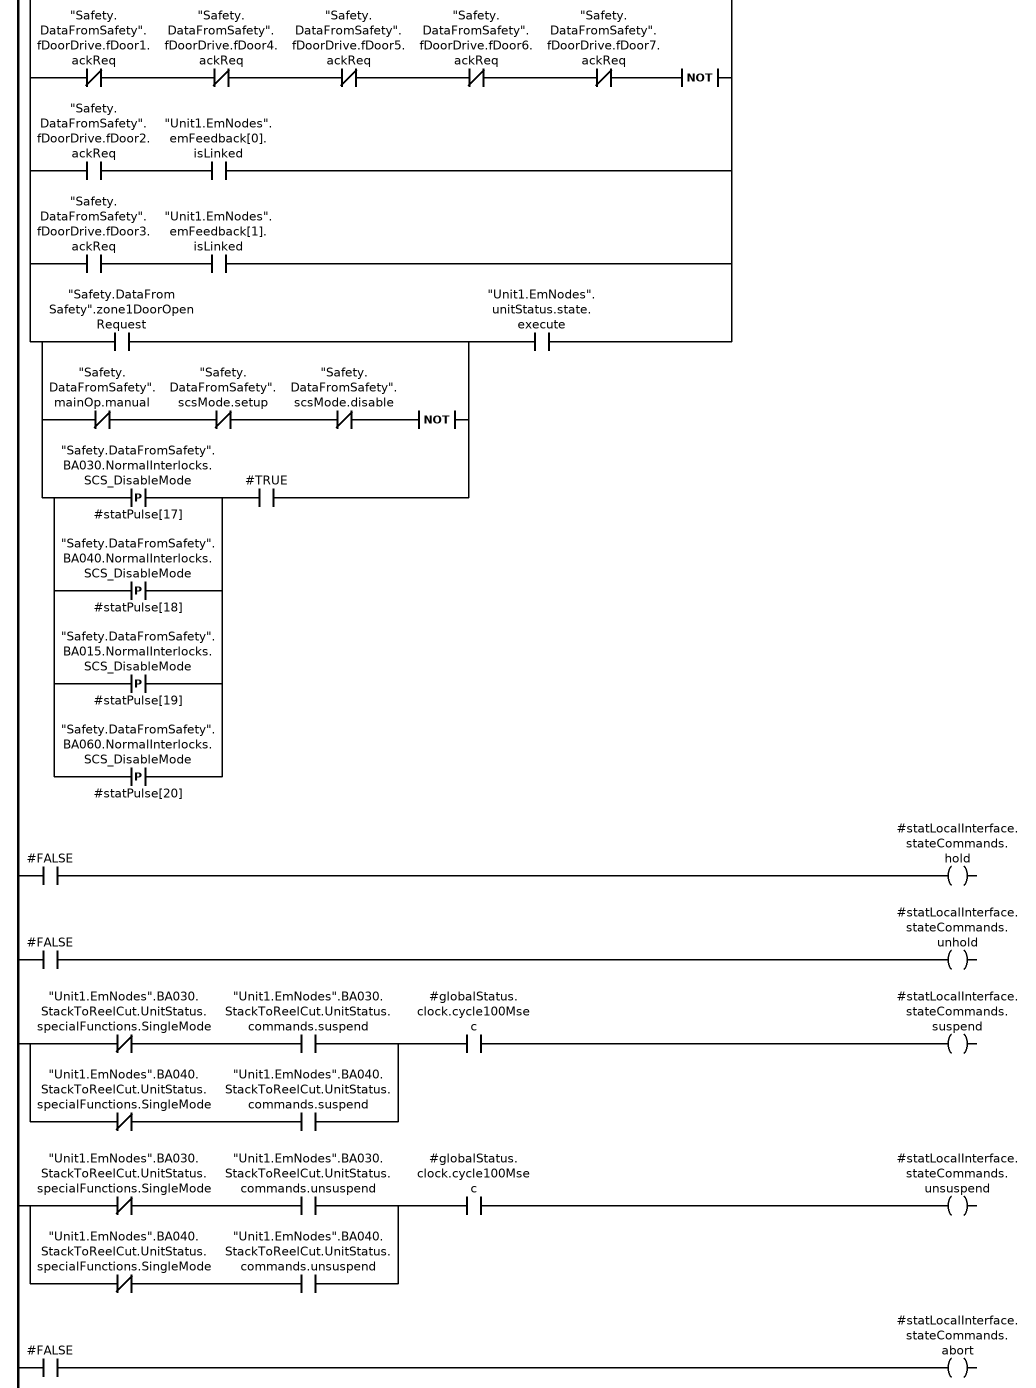
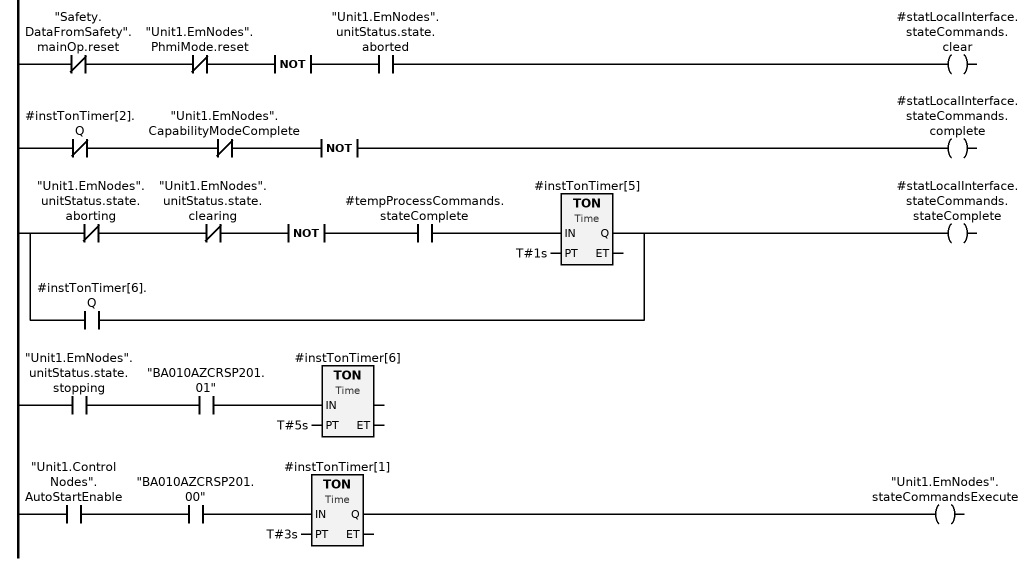
   RUNG wire#powerrail
      Contact( "Safety.DataFromSafety".mainOp.auto )
      Contact( #globalStatus.clock.cycle100Msec )
      I_Contact( #statLocalInterface.modeRequests.userMode01 )
      I_Contact( #instTonTimer[7].Q )
      I_Contact( "Unit1.EmNodes".WakeupRecoveryRequired )
      Coil( #statLocalInterface.modeRequests.production )
   END_RUNG
   RUNG wire#powerrail
      Contact( "Safety.DataFromSafety".mainOp.manual )
      Contact( "Safety.DataFromSafety".scsMode.setup )
      Contact( #globalStatus.clock.cycle100Msec )
      I_Contact( #statLocalInterface.modeRequests.userMode01 )
      I_Contact( #instTonTimer[7].Q )
      I_Contact( "Unit1.EmNodes".WakeupRecoveryRequired )
      Coil( #statLocalInterface.modeRequests.maintenance )
   END_RUNG
   RUNG wire#powerrail
      Contact( "Safety.DataFromSafety".mainOp.manual )
      Contact( "Safety.DataFromSafety".scsMode.auto )
      Contact( #globalStatus.clock.cycle100Msec )
      I_Contact( #statLocalInterface.modeRequests.userMode01 )
      I_Contact( #instTonTimer[7].Q )
      I_Contact( "Unit1.EmNodes".WakeupRecoveryRequired )
      Coil( #statLocalInterface.modeRequests.manual )
   END_RUNG
   RUNG wire#powerrail
      I_Contact( "Safety.DataFromSafety".scsMode.disable )
      Contact( "Unit1.EmNodes".Z_FOLD_AllEstopsOK )
      Not()
      wire#w1
      I_Contact( #globalStatus.activateSimulation )
      { S7_Templates := "time_type := Time" } #instTonTimer[7].TON(pt := T#200ms, et =>)
      Contact( #globalStatus.clock.cycle100Msec )
      Coil( #statLocalInterface.modeRequests.userMode01 )
   END_RUNG
   RUNG wire#powerrail
      Contact( "Unit1.EmNodes".Zone1SafetyStatus.MFDoorOpen )
   END_RUNG wire#w1
   RUNG wire#powerrail
      I_Contact( "Unit1.EmNodes".Zone1SafetyStatus.safetyReleased1 )
      I_Contact( "Unit1.EmNodes".Zone1SafetyStatus.safetyReleased2 )
   END_RUNG wire#w1
   RUNG wire#powerrail
      I_Contact( "Unit1.EmNodes".Zone2SafetyStatus.safetyReleased1 )
      I_Contact( "Unit1.EmNodes".Zone2SafetyStatus.safetyReleased2 )
      Contact( "Unit1.EmNodes".emFeedback[0].isLinked )
   END_RUNG wire#w1
   RUNG wire#powerrail
      I_Contact( "Unit1.EmNodes".Zone3SafetyStatus.safetyReleased1 )
      I_Contact( "Unit1.EmNodes".Zone3SafetyStatus.safetyReleased2 )
      Contact( "Unit1.EmNodes".emFeedback[1].isLinked )
   END_RUNG wire#w1
   RUNG wire#powerrail
      Contact( "Unit1.EmNodes".SleepModeChangeReq )
      Contact( #globalStatus.clock.cycle100Msec )
      Coil( #statLocalInterface.modeRequests.userMode02 )
   END_RUNG
   RUNG wire#powerrail
      Contact( "Unit1.EmNodes".DeepSleepModeChangeReq )
      Contact( #globalStatus.clock.cycle100Msec )
      Coil( #statLocalInterface.modeRequests.userMode03 )
   END_RUNG
   RUNG wire#powerrail
      I_Contact( "Safety.DataFromSafety".mainOp.reset )
      I_Contact( "Unit1.EmNodes".PhmiMode.reset )
      Not()
      I_Contact( "Unit1.EmNodes".unitStatus.state.aborted )
      Coil( #statLocalInterface.stateCommands.reset )
   END_RUNG
   RUNG wire#powerrail
      P_Contact(operand := "Safety.DataFromSafety".mainOp.home, bit := #statPulse[16])
      Contact( "Unit1.ControlNodes".InitializeEnable )
      wire#w2
      I_Contact( "Unit1.EmNodes".unitStatus.state.starting )
      I_Contact( "Unit1.EmNodes".unitStatus.state.stopped )
      I_Contact( "Unit1.EmNodes".unitStatus.state.aborted )
      Coil( #statLocalInterface.stateCommands.start )
   END_RUNG
   RUNG wire#powerrail
      Contact( #statLocalInterface.stateCommands.start )
   END_RUNG wire#w2
   RUNG wire#powerrail
      Contact( "BA010AZCRSP201.01" )
      wire#w3
      I_Contact( "Unit1.EmNodes".unitStatus.state.stopped )
      Coil( #statLocalInterface.stateCommands.stop )
   END_RUNG
   RUNG wire#powerrail
      I_Contact( "Unit1.EmNodes".BA030.StackToReelCut.UnitStatus.commands.stop )
      I_Contact( "Unit1.EmNodes".BA040.StackToReelCut.UnitStatus.commands.stop )
      Not()
   END_RUNG wire#w3
   RUNG wire#powerrail
      I_Contact( "Safety.DataFromSafety".fDoorDrive.fDoor1.ackReq )
      I_Contact( "Safety.DataFromSafety".fDoorDrive.fDoor4.ackReq )
      I_Contact( "Safety.DataFromSafety".fDoorDrive.fDoor5.ackReq )
      I_Contact( "Safety.DataFromSafety".fDoorDrive.fDoor6.ackReq )
      I_Contact( "Safety.DataFromSafety".fDoorDrive.fDoor7.ackReq )
      Not()
   END_RUNG wire#w3
   RUNG wire#powerrail
      Contact( "Safety.DataFromSafety".fDoorDrive.fDoor2.ackReq )
      Contact( "Unit1.EmNodes".emFeedback[0].isLinked )
   END_RUNG wire#w3
   RUNG wire#powerrail
      Contact( "Safety.DataFromSafety".fDoorDrive.fDoor3.ackReq )
      Contact( "Unit1.EmNodes".emFeedback[1].isLinked )
   END_RUNG wire#w3
   RUNG wire#powerrail
      Contact( "Safety.DataFromSafety".zone1DoorOpenRequest )
      wire#w4
      Contact( "Unit1.EmNodes".unitStatus.state.execute )
   END_RUNG wire#w3
   RUNG wire#powerrail
      I_Contact( "Safety.DataFromSafety".mainOp.manual )
      I_Contact( "Safety.DataFromSafety".scsMode.setup )
      I_Contact( "Safety.DataFromSafety".scsMode.disable )
      Not()
   END_RUNG wire#w4
   RUNG wire#powerrail
      P_Contact(operand := "Safety.DataFromSafety".BA030.NormalInterlocks.SCS_DisableMode, bit := #statPulse[17])
      wire#w5
      Contact( #TRUE )
   END_RUNG wire#w4
   RUNG wire#powerrail
      P_Contact(operand := "Safety.DataFromSafety".BA040.NormalInterlocks.SCS_DisableMode, bit := #statPulse[18])
   END_RUNG wire#w5
   RUNG wire#powerrail
      P_Contact(operand := "Safety.DataFromSafety".BA015.NormalInterlocks.SCS_DisableMode, bit := #statPulse[19])
   END_RUNG wire#w5
   RUNG wire#powerrail
      P_Contact(operand := "Safety.DataFromSafety".BA060.NormalInterlocks.SCS_DisableMode, bit := #statPulse[20])
   END_RUNG wire#w5
   RUNG wire#powerrail
      Contact( #FALSE )
      Coil( #statLocalInterface.stateCommands.hold )
   END_RUNG
   RUNG wire#powerrail
      Contact( #FALSE )
      Coil( #statLocalInterface.stateCommands.unhold )
   END_RUNG
   RUNG wire#powerrail
      I_Contact( "Unit1.EmNodes".BA030.StackToReelCut.UnitStatus.specialFunctions.SingleMode )
      Contact( "Unit1.EmNodes".BA030.StackToReelCut.UnitStatus.commands.suspend )
      wire#w6
      Contact( #globalStatus.clock.cycle100Msec )
      Coil( #statLocalInterface.stateCommands.suspend )
   END_RUNG
   RUNG wire#powerrail
      I_Contact( "Unit1.EmNodes".BA040.StackToReelCut.UnitStatus.specialFunctions.SingleMode )
      Contact( "Unit1.EmNodes".BA040.StackToReelCut.UnitStatus.commands.suspend )
   END_RUNG wire#w6
   RUNG wire#powerrail
      I_Contact( "Unit1.EmNodes".BA030.StackToReelCut.UnitStatus.specialFunctions.SingleMode )
      Contact( "Unit1.EmNodes".BA030.StackToReelCut.UnitStatus.commands.unsuspend )
      wire#w7
      Contact( #globalStatus.clock.cycle100Msec )
      Coil( #statLocalInterface.stateCommands.unsuspend )
   END_RUNG
   RUNG wire#powerrail
      I_Contact( "Unit1.EmNodes".BA040.StackToReelCut.UnitStatus.specialFunctions.SingleMode )
      Contact( "Unit1.EmNodes".BA040.StackToReelCut.UnitStatus.commands.unsuspend )
   END_RUNG wire#w7
   RUNG wire#powerrail
      Contact( #FALSE )
      Coil( #statLocalInterface.stateCommands.abort )
   END_RUNG
   RUNG wire#powerrail
      I_Contact( "Safety.DataFromSafety".mainOp.reset )
      I_Contact( "Unit1.EmNodes".PhmiMode.reset )
      Not()
      Contact( "Unit1.EmNodes".unitStatus.state.aborted )
      Coil( #statLocalInterface.stateCommands.clear )
   END_RUNG
   RUNG wire#powerrail
      I_Contact( #instTonTimer[2].Q )
      I_Contact( "Unit1.EmNodes".CapabilityModeComplete )
      Not()
      Coil( #statLocalInterface.stateCommands.complete )
   END_RUNG
   RUNG wire#powerrail
      I_Contact( "Unit1.EmNodes".unitStatus.state.aborting )
      I_Contact( "Unit1.EmNodes".unitStatus.state.clearing )
      Not()
      Contact( #tempProcessCommands.stateComplete )
      { S7_Templates := "time_type := Time" } #instTonTimer[5].TON(pt := T#1s, et =>)
      wire#w8
      Coil( #statLocalInterface.stateCommands.stateComplete )
   END_RUNG
   RUNG wire#powerrail
      Contact( #instTonTimer[6].Q )
   END_RUNG wire#w8
   RUNG wire#powerrail
      Contact( "Unit1.EmNodes".unitStatus.state.stopping )
      Contact( "BA010AZCRSP201.01" )
      { S7_Templates := "time_type := Time" } #instTonTimer[6].TON(pt := T#5s, et =>)
   END_RUNG
   RUNG wire#powerrail
      Contact( "Unit1.ControlNodes".AutoStartEnable )
      Contact( "BA010AZCRSP201.00" )
      { S7_Templates := "time_type := Time" } #instTonTimer[1].TON(pt := T#3s, et =>)
      Coil( "Unit1.EmNodes".stateCommandsExecute )
   END_RUNG
   // the same network as SCL:
   #statLocalInterface.modeRequests.production := "Safety.DataFromSafety".mainOp.auto AND #globalStatus.clock.cycle100Msec AND NOT #statLocalInterface.modeRequests.userMode01 AND NOT #instTonTimer[7].Q AND NOT "Unit1.EmNodes".WakeupRecoveryRequired;
   #statLocalInterface.modeRequests.maintenance := "Safety.DataFromSafety".mainOp.manual AND "Safety.DataFromSafety".scsMode.setup AND #globalStatus.clock.cycle100Msec AND NOT #statLocalInterface.modeRequests.userMode01 AND NOT #instTonTimer[7].Q AND NOT "Unit1.EmNodes".WakeupRecoveryRequired;
   #statLocalInterface.modeRequests.manual := "Safety.DataFromSafety".mainOp.manual AND "Safety.DataFromSafety".scsMode.auto AND #globalStatus.clock.cycle100Msec AND NOT #statLocalInterface.modeRequests.userMode01 AND NOT #instTonTimer[7].Q AND NOT "Unit1.EmNodes".WakeupRecoveryRequired;
   #instTonTimer[7].TON(IN := (NOT (NOT "Safety.DataFromSafety".scsMode.disable AND "Unit1.EmNodes".Z_FOLD_AllEstopsOK) OR "Unit1.EmNodes".Zone1SafetyStatus.MFDoorOpen OR (NOT "Unit1.EmNodes".Zone1SafetyStatus.safetyReleased1 AND NOT "Unit1.EmNodes".Zone1SafetyStatus.safetyReleased2) OR (NOT "Unit1.EmNodes".Zone2SafetyStatus.safetyReleased1 AND NOT "Unit1.EmNodes".Zone2SafetyStatus.safetyReleased2 AND "Unit1.EmNodes".emFeedback[0].isLinked) OR (NOT "Unit1.EmNodes".Zone3SafetyStatus.safetyReleased1 AND NOT "Unit1.EmNodes".Zone3SafetyStatus.safetyReleased2 AND "Unit1.EmNodes".emFeedback[1].isLinked)) AND NOT #globalStatus.activateSimulation,
                        PT := T#200ms);
   #statLocalInterface.modeRequests.userMode01 := #instTonTimer[7].Q AND #globalStatus.clock.cycle100Msec;
   #statLocalInterface.modeRequests.userMode02 := "Unit1.EmNodes".SleepModeChangeReq AND #globalStatus.clock.cycle100Msec;
   #statLocalInterface.modeRequests.userMode03 := "Unit1.EmNodes".DeepSleepModeChangeReq AND #globalStatus.clock.cycle100Msec;
   #statLocalInterface.stateCommands.reset := NOT (NOT "Safety.DataFromSafety".mainOp.reset AND NOT "Unit1.EmNodes".PhmiMode.reset) AND NOT "Unit1.EmNodes".unitStatus.state.aborted;
   #_w1 := "Safety.DataFromSafety".mainOp.home AND NOT #statPulse[16];   // rising edge of "Safety.DataFromSafety".mainOp.home
   #statPulse[16] := "Safety.DataFromSafety".mainOp.home;
   #statLocalInterface.stateCommands.start := ((#_w1 AND "Unit1.ControlNodes".InitializeEnable) OR #statLocalInterface.stateCommands.start) AND NOT "Unit1.EmNodes".unitStatus.state.starting AND NOT "Unit1.EmNodes".unitStatus.state.stopped AND NOT "Unit1.EmNodes".unitStatus.state.aborted;
   #_w2 := "Safety.DataFromSafety".BA030.NormalInterlocks.SCS_DisableMode AND NOT #statPulse[17];   // rising edge of "Safety.DataFromSafety".BA030.NormalInterlocks.SCS_DisableMode
   #statPulse[17] := "Safety.DataFromSafety".BA030.NormalInterlocks.SCS_DisableMode;
   #_w3 := "Safety.DataFromSafety".BA040.NormalInterlocks.SCS_DisableMode AND NOT #statPulse[18];   // rising edge of "Safety.DataFromSafety".BA040.NormalInterlocks.SCS_DisableMode
   #statPulse[18] := "Safety.DataFromSafety".BA040.NormalInterlocks.SCS_DisableMode;
   #_w4 := "Safety.DataFromSafety".BA015.NormalInterlocks.SCS_DisableMode AND NOT #statPulse[19];   // rising edge of "Safety.DataFromSafety".BA015.NormalInterlocks.SCS_DisableMode
   #statPulse[19] := "Safety.DataFromSafety".BA015.NormalInterlocks.SCS_DisableMode;
   #_w5 := "Safety.DataFromSafety".BA060.NormalInterlocks.SCS_DisableMode AND NOT #statPulse[20];   // rising edge of "Safety.DataFromSafety".BA060.NormalInterlocks.SCS_DisableMode
   #statPulse[20] := "Safety.DataFromSafety".BA060.NormalInterlocks.SCS_DisableMode;
   #statLocalInterface.stateCommands.stop := ("BA010AZCRSP201.01" OR NOT (NOT "Unit1.EmNodes".BA030.StackToReelCut.UnitStatus.commands.stop AND NOT "Unit1.EmNodes".BA040.StackToReelCut.UnitStatus.commands.stop) OR NOT (NOT "Safety.DataFromSafety".fDoorDrive.fDoor1.ackReq AND NOT "Safety.DataFromSafety".fDoorDrive.fDoor4.ackReq AND NOT "Safety.DataFromSafety".fDoorDrive.fDoor5.ackReq AND NOT "Safety.DataFromSafety".fDoorDrive.fDoor6.ackReq AND NOT "Safety.DataFromSafety".fDoorDrive.fDoor7.ackReq) OR ("Safety.DataFromSafety".fDoorDrive.fDoor2.ackReq AND "Unit1.EmNodes".emFeedback[0].isLinked) OR ("Safety.DataFromSafety".fDoorDrive.fDoor3.ackReq AND "Unit1.EmNodes".emFeedback[1].isLinked) OR (("Safety.DataFromSafety".zone1DoorOpenRequest OR NOT (NOT "Safety.DataFromSafety".mainOp.manual AND NOT "Safety.DataFromSafety".scsMode.setup AND NOT "Safety.DataFromSafety".scsMode.disable) OR ((#_w2 OR #_w3 OR #_w4 OR #_w5) AND #TRUE)) AND "Unit1.EmNodes".unitStatus.state.execute)) AND NOT "Unit1.EmNodes".unitStatus.state.stopped;
   #statLocalInterface.stateCommands.hold := #FALSE;
   #statLocalInterface.stateCommands.unhold := #FALSE;
   #statLocalInterface.stateCommands.suspend := ((NOT "Unit1.EmNodes".BA030.StackToReelCut.UnitStatus.specialFunctions.SingleMode AND "Unit1.EmNodes".BA030.StackToReelCut.UnitStatus.commands.suspend) OR (NOT "Unit1.EmNodes".BA040.StackToReelCut.UnitStatus.specialFunctions.SingleMode AND "Unit1.EmNodes".BA040.StackToReelCut.UnitStatus.commands.suspend)) AND #globalStatus.clock.cycle100Msec;
   #statLocalInterface.stateCommands.unsuspend := ((NOT "Unit1.EmNodes".BA030.StackToReelCut.UnitStatus.specialFunctions.SingleMode AND "Unit1.EmNodes".BA030.StackToReelCut.UnitStatus.commands.unsuspend) OR (NOT "Unit1.EmNodes".BA040.StackToReelCut.UnitStatus.specialFunctions.SingleMode AND "Unit1.EmNodes".BA040.StackToReelCut.UnitStatus.commands.unsuspend)) AND #globalStatus.clock.cycle100Msec;
   #statLocalInterface.stateCommands.abort := #FALSE;
   #statLocalInterface.stateCommands.clear := NOT (NOT "Safety.DataFromSafety".mainOp.reset AND NOT "Unit1.EmNodes".PhmiMode.reset) AND "Unit1.EmNodes".unitStatus.state.aborted;
   #statLocalInterface.stateCommands.complete := NOT (NOT #instTonTimer[2].Q AND NOT "Unit1.EmNodes".CapabilityModeComplete);
   #instTonTimer[5].TON(IN := NOT (NOT "Unit1.EmNodes".unitStatus.state.aborting AND NOT "Unit1.EmNodes".unitStatus.state.clearing) AND #tempProcessCommands.stateComplete,
                        PT := T#1s);
   #statLocalInterface.stateCommands.stateComplete := #instTonTimer[5].Q OR #instTonTimer[6].Q;
   #instTonTimer[6].TON(IN := "Unit1.EmNodes".unitStatus.state.stopping AND "BA010AZCRSP201.01", PT := T#5s);
   #instTonTimer[1].TON(IN := "Unit1.ControlNodes".AutoStartEnable AND "BA010AZCRSP201.00", PT := T#3s);
   "Unit1.EmNodes".stateCommandsExecute := #instTonTimer[1].Q;
END_REGION

REGION Network 40: Main Op Lamp
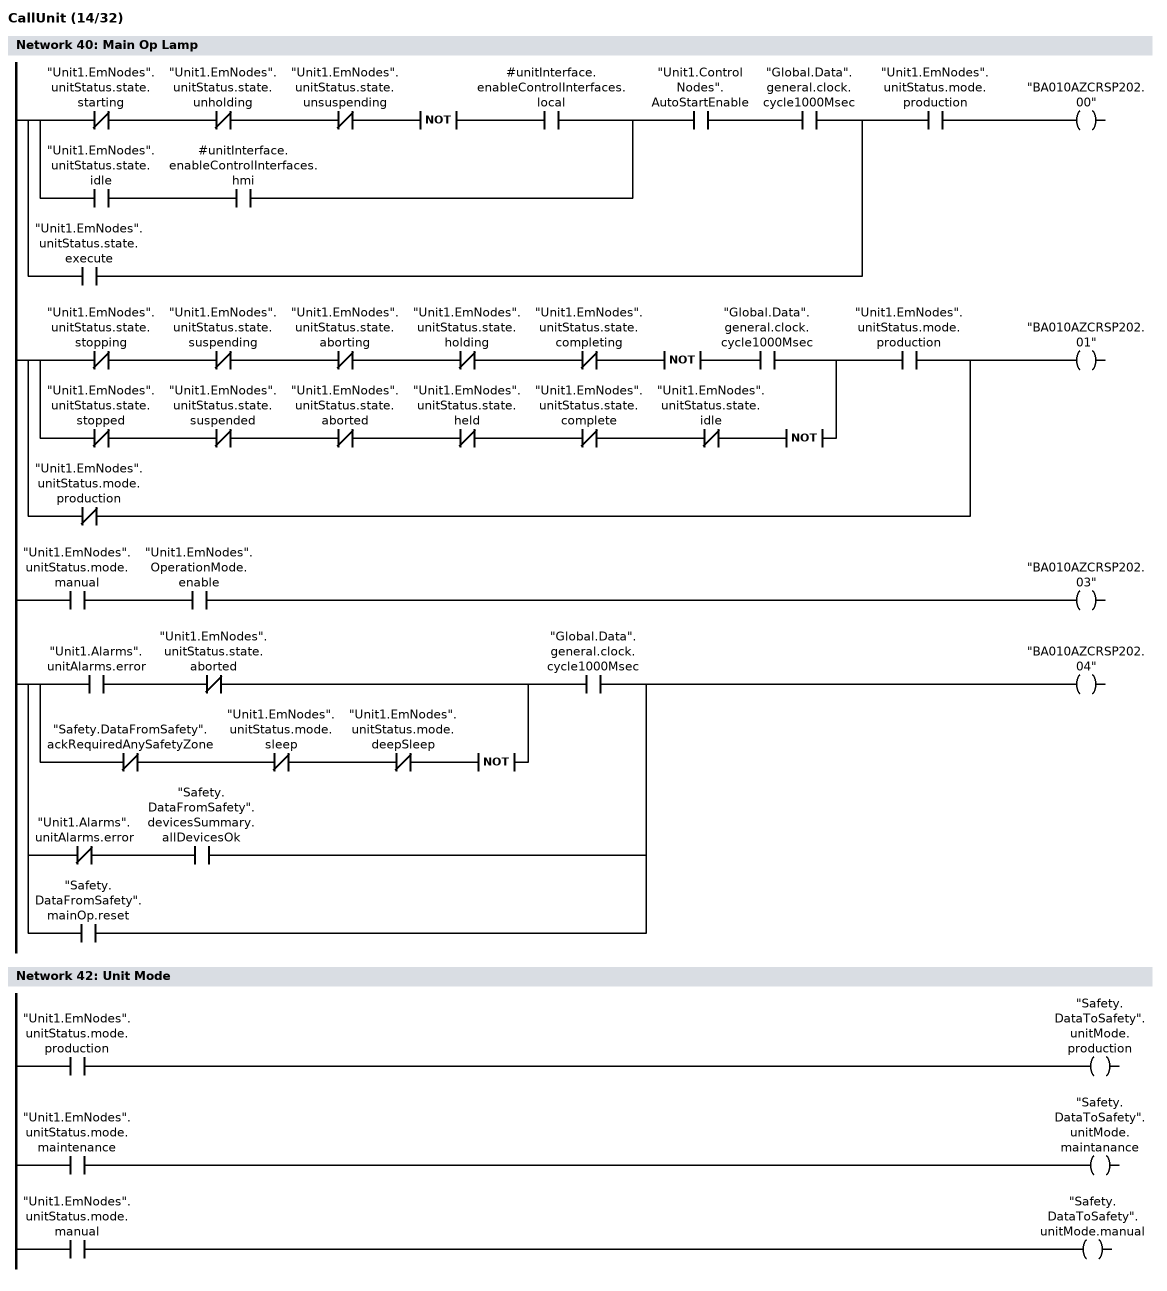
   RUNG wire#powerrail
      I_Contact( "Unit1.EmNodes".unitStatus.state.starting )
      I_Contact( "Unit1.EmNodes".unitStatus.state.unholding )
      I_Contact( "Unit1.EmNodes".unitStatus.state.unsuspending )
      Not()
      Contact( #unitInterface.enableControlInterfaces.local )
      wire#w1
      Contact( "Unit1.ControlNodes".AutoStartEnable )
      Contact( "Global.Data".general.clock.cycle1000Msec )
      wire#w2
      Contact( "Unit1.EmNodes".unitStatus.mode.production )
      Coil( "BA010AZCRSP202.00" )
   END_RUNG
   RUNG wire#powerrail
      Contact( "Unit1.EmNodes".unitStatus.state.idle )
      Contact( #unitInterface.enableControlInterfaces.hmi )
   END_RUNG wire#w1
   RUNG wire#powerrail
      Contact( "Unit1.EmNodes".unitStatus.state.execute )
   END_RUNG wire#w2
   RUNG wire#powerrail
      I_Contact( "Unit1.EmNodes".unitStatus.state.stopping )
      I_Contact( "Unit1.EmNodes".unitStatus.state.suspending )
      I_Contact( "Unit1.EmNodes".unitStatus.state.aborting )
      I_Contact( "Unit1.EmNodes".unitStatus.state.holding )
      I_Contact( "Unit1.EmNodes".unitStatus.state.completing )
      Not()
      Contact( "Global.Data".general.clock.cycle1000Msec )
      wire#w3
      Contact( "Unit1.EmNodes".unitStatus.mode.production )
      wire#w4
      Coil( "BA010AZCRSP202.01" )
   END_RUNG
   RUNG wire#powerrail
      I_Contact( "Unit1.EmNodes".unitStatus.state.stopped )
      I_Contact( "Unit1.EmNodes".unitStatus.state.suspended )
      I_Contact( "Unit1.EmNodes".unitStatus.state.aborted )
      I_Contact( "Unit1.EmNodes".unitStatus.state.held )
      I_Contact( "Unit1.EmNodes".unitStatus.state.complete )
      I_Contact( "Unit1.EmNodes".unitStatus.state.idle )
      Not()
   END_RUNG wire#w3
   RUNG wire#powerrail
      I_Contact( "Unit1.EmNodes".unitStatus.mode.production )
   END_RUNG wire#w4
   RUNG wire#powerrail
      Contact( "Unit1.EmNodes".unitStatus.mode.manual )
      Contact( "Unit1.EmNodes".OperationMode.enable )
      Coil( "BA010AZCRSP202.03" )
   END_RUNG
   RUNG wire#powerrail
      Contact( "Unit1.Alarms".unitAlarms.error )
      I_Contact( "Unit1.EmNodes".unitStatus.state.aborted )
      wire#w5
      Contact( "Global.Data".general.clock.cycle1000Msec )
      wire#w6
      Coil( "BA010AZCRSP202.04" )
   END_RUNG
   RUNG wire#powerrail
      I_Contact( "Safety.DataFromSafety".ackRequiredAnySafetyZone )
      I_Contact( "Unit1.EmNodes".unitStatus.mode.sleep )
      I_Contact( "Unit1.EmNodes".unitStatus.mode.deepSleep )
      Not()
   END_RUNG wire#w5
   RUNG wire#powerrail
      I_Contact( "Unit1.Alarms".unitAlarms.error )
      Contact( "Safety.DataFromSafety".devicesSummary.allDevicesOk )
   END_RUNG wire#w6
   RUNG wire#powerrail
      Contact( "Safety.DataFromSafety".mainOp.reset )
   END_RUNG wire#w6
   // the same network as SCL:
   "BA010AZCRSP202.00" := ((((NOT (NOT "Unit1.EmNodes".unitStatus.state.starting AND NOT "Unit1.EmNodes".unitStatus.state.unholding AND NOT "Unit1.EmNodes".unitStatus.state.unsuspending) AND #unitInterface.enableControlInterfaces.local) OR ("Unit1.EmNodes".unitStatus.state.idle AND #unitInterface.enableControlInterfaces.hmi)) AND "Unit1.ControlNodes".AutoStartEnable AND "Global.Data".general.clock.cycle1000Msec) OR "Unit1.EmNodes".unitStatus.state.execute) AND "Unit1.EmNodes".unitStatus.mode.production;
   "BA010AZCRSP202.01" := (((NOT (NOT "Unit1.EmNodes".unitStatus.state.stopping AND NOT "Unit1.EmNodes".unitStatus.state.suspending AND NOT "Unit1.EmNodes".unitStatus.state.aborting AND NOT "Unit1.EmNodes".unitStatus.state.holding AND NOT "Unit1.EmNodes".unitStatus.state.completing) AND "Global.Data".general.clock.cycle1000Msec) OR NOT (NOT "Unit1.EmNodes".unitStatus.state.stopped AND NOT "Unit1.EmNodes".unitStatus.state.suspended AND NOT "Unit1.EmNodes".unitStatus.state.aborted AND NOT "Unit1.EmNodes".unitStatus.state.held AND NOT "Unit1.EmNodes".unitStatus.state.complete AND NOT "Unit1.EmNodes".unitStatus.state.idle)) AND "Unit1.EmNodes".unitStatus.mode.production) OR NOT "Unit1.EmNodes".unitStatus.mode.production;
   "BA010AZCRSP202.03" := "Unit1.EmNodes".unitStatus.mode.manual AND "Unit1.EmNodes".OperationMode.enable;
   "BA010AZCRSP202.04" := ((("Unit1.Alarms".unitAlarms.error AND NOT "Unit1.EmNodes".unitStatus.state.aborted) OR NOT (NOT "Safety.DataFromSafety".ackRequiredAnySafetyZone AND NOT "Unit1.EmNodes".unitStatus.mode.sleep AND NOT "Unit1.EmNodes".unitStatus.mode.deepSleep)) AND "Global.Data".general.clock.cycle1000Msec) OR (NOT "Unit1.Alarms".unitAlarms.error AND "Safety.DataFromSafety".devicesSummary.allDevicesOk) OR "Safety.DataFromSafety".mainOp.reset;
END_REGION

REGION Network 41: ******************** Data To Safety Mapping ********************
END_REGION

REGION Network 42: Unit Mode
   RUNG wire#powerrail
      Contact( "Unit1.EmNodes".unitStatus.mode.production )
      Coil( "Safety.DataToSafety".unitMode.production )
   END_RUNG
   RUNG wire#powerrail
      Contact( "Unit1.EmNodes".unitStatus.mode.maintenance )
      Coil( "Safety.DataToSafety".unitMode.maintanance )
   END_RUNG
   RUNG wire#powerrail
      Contact( "Unit1.EmNodes".unitStatus.mode.manual )
      Coil( "Safety.DataToSafety".unitMode.manual )
   END_RUNG
   // the same network as SCL:
   "Safety.DataToSafety".unitMode.production := "Unit1.EmNodes".unitStatus.mode.production;
   "Safety.DataToSafety".unitMode.maintanance := "Unit1.EmNodes".unitStatus.mode.maintenance;
   "Safety.DataToSafety".unitMode.manual := "Unit1.EmNodes".unitStatus.mode.manual;
END_REGION

REGION Network 43: Unit States
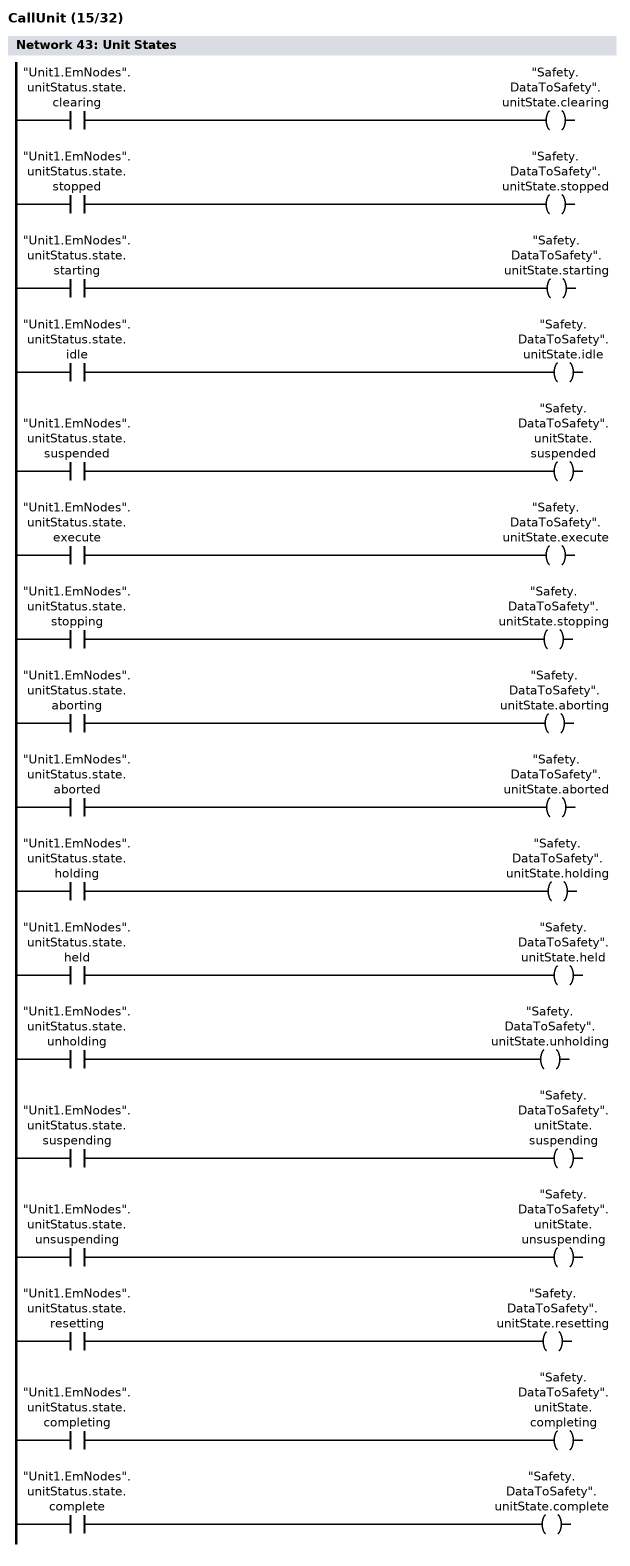
   RUNG wire#powerrail
      Contact( "Unit1.EmNodes".unitStatus.state.clearing )
      Coil( "Safety.DataToSafety".unitState.clearing )
   END_RUNG
   RUNG wire#powerrail
      Contact( "Unit1.EmNodes".unitStatus.state.stopped )
      Coil( "Safety.DataToSafety".unitState.stopped )
   END_RUNG
   RUNG wire#powerrail
      Contact( "Unit1.EmNodes".unitStatus.state.starting )
      Coil( "Safety.DataToSafety".unitState.starting )
   END_RUNG
   RUNG wire#powerrail
      Contact( "Unit1.EmNodes".unitStatus.state.idle )
      Coil( "Safety.DataToSafety".unitState.idle )
   END_RUNG
   RUNG wire#powerrail
      Contact( "Unit1.EmNodes".unitStatus.state.suspended )
      Coil( "Safety.DataToSafety".unitState.suspended )
   END_RUNG
   RUNG wire#powerrail
      Contact( "Unit1.EmNodes".unitStatus.state.execute )
      Coil( "Safety.DataToSafety".unitState.execute )
   END_RUNG
   RUNG wire#powerrail
      Contact( "Unit1.EmNodes".unitStatus.state.stopping )
      Coil( "Safety.DataToSafety".unitState.stopping )
   END_RUNG
   RUNG wire#powerrail
      Contact( "Unit1.EmNodes".unitStatus.state.aborting )
      Coil( "Safety.DataToSafety".unitState.aborting )
   END_RUNG
   RUNG wire#powerrail
      Contact( "Unit1.EmNodes".unitStatus.state.aborted )
      Coil( "Safety.DataToSafety".unitState.aborted )
   END_RUNG
   RUNG wire#powerrail
      Contact( "Unit1.EmNodes".unitStatus.state.holding )
      Coil( "Safety.DataToSafety".unitState.holding )
   END_RUNG
   RUNG wire#powerrail
      Contact( "Unit1.EmNodes".unitStatus.state.held )
      Coil( "Safety.DataToSafety".unitState.held )
   END_RUNG
   RUNG wire#powerrail
      Contact( "Unit1.EmNodes".unitStatus.state.unholding )
      Coil( "Safety.DataToSafety".unitState.unholding )
   END_RUNG
   RUNG wire#powerrail
      Contact( "Unit1.EmNodes".unitStatus.state.suspending )
      Coil( "Safety.DataToSafety".unitState.suspending )
   END_RUNG
   RUNG wire#powerrail
      Contact( "Unit1.EmNodes".unitStatus.state.unsuspending )
      Coil( "Safety.DataToSafety".unitState.unsuspending )
   END_RUNG
   RUNG wire#powerrail
      Contact( "Unit1.EmNodes".unitStatus.state.resetting )
      Coil( "Safety.DataToSafety".unitState.resetting )
   END_RUNG
   RUNG wire#powerrail
      Contact( "Unit1.EmNodes".unitStatus.state.completing )
      Coil( "Safety.DataToSafety".unitState.completing )
   END_RUNG
   RUNG wire#powerrail
      Contact( "Unit1.EmNodes".unitStatus.state.complete )
      Coil( "Safety.DataToSafety".unitState.complete )
   END_RUNG
   // the same network as SCL:
   "Safety.DataToSafety".unitState.clearing := "Unit1.EmNodes".unitStatus.state.clearing;
   "Safety.DataToSafety".unitState.stopped := "Unit1.EmNodes".unitStatus.state.stopped;
   "Safety.DataToSafety".unitState.starting := "Unit1.EmNodes".unitStatus.state.starting;
   "Safety.DataToSafety".unitState.idle := "Unit1.EmNodes".unitStatus.state.idle;
   "Safety.DataToSafety".unitState.suspended := "Unit1.EmNodes".unitStatus.state.suspended;
   "Safety.DataToSafety".unitState.execute := "Unit1.EmNodes".unitStatus.state.execute;
   "Safety.DataToSafety".unitState.stopping := "Unit1.EmNodes".unitStatus.state.stopping;
   "Safety.DataToSafety".unitState.aborting := "Unit1.EmNodes".unitStatus.state.aborting;
   "Safety.DataToSafety".unitState.aborted := "Unit1.EmNodes".unitStatus.state.aborted;
   "Safety.DataToSafety".unitState.holding := "Unit1.EmNodes".unitStatus.state.holding;
   "Safety.DataToSafety".unitState.held := "Unit1.EmNodes".unitStatus.state.held;
   "Safety.DataToSafety".unitState.unholding := "Unit1.EmNodes".unitStatus.state.unholding;
   "Safety.DataToSafety".unitState.suspending := "Unit1.EmNodes".unitStatus.state.suspending;
   "Safety.DataToSafety".unitState.unsuspending := "Unit1.EmNodes".unitStatus.state.unsuspending;
   "Safety.DataToSafety".unitState.resetting := "Unit1.EmNodes".unitStatus.state.resetting;
   "Safety.DataToSafety".unitState.completing := "Unit1.EmNodes".unitStatus.state.completing;
   "Safety.DataToSafety".unitState.complete := "Unit1.EmNodes".unitStatus.state.complete;
END_REGION

REGION Network 44: Unwinder Link
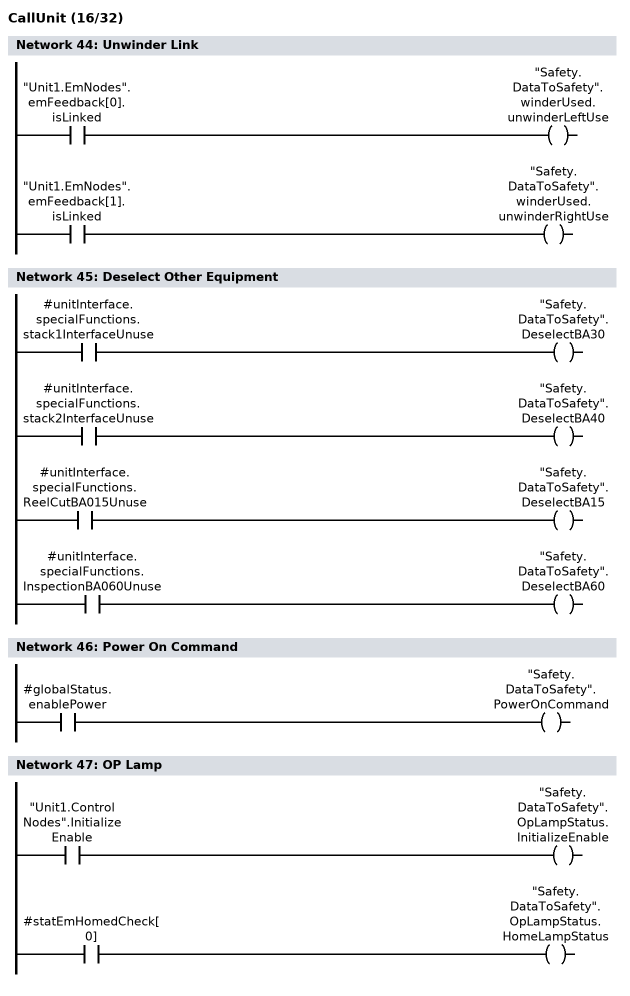
   RUNG wire#powerrail
      Contact( "Unit1.EmNodes".emFeedback[0].isLinked )
      Coil( "Safety.DataToSafety".winderUsed.unwinderLeftUse )
   END_RUNG
   RUNG wire#powerrail
      Contact( "Unit1.EmNodes".emFeedback[1].isLinked )
      Coil( "Safety.DataToSafety".winderUsed.unwinderRightUse )
   END_RUNG
   // the same network as SCL:
   "Safety.DataToSafety".winderUsed.unwinderLeftUse := "Unit1.EmNodes".emFeedback[0].isLinked;
   "Safety.DataToSafety".winderUsed.unwinderRightUse := "Unit1.EmNodes".emFeedback[1].isLinked;
END_REGION

REGION Network 45: Deselect Other Equipment
   RUNG wire#powerrail
      Contact( #unitInterface.specialFunctions.stack1InterfaceUnuse )
      Coil( "Safety.DataToSafety".DeselectBA30 )
   END_RUNG
   RUNG wire#powerrail
      Contact( #unitInterface.specialFunctions.stack2InterfaceUnuse )
      Coil( "Safety.DataToSafety".DeselectBA40 )
   END_RUNG
   RUNG wire#powerrail
      Contact( #unitInterface.specialFunctions.ReelCutBA015Unuse )
      Coil( "Safety.DataToSafety".DeselectBA15 )
   END_RUNG
   RUNG wire#powerrail
      Contact( #unitInterface.specialFunctions.InspectionBA060Unuse )
      Coil( "Safety.DataToSafety".DeselectBA60 )
   END_RUNG
   // the same network as SCL:
   "Safety.DataToSafety".DeselectBA30 := #unitInterface.specialFunctions.stack1InterfaceUnuse;
   "Safety.DataToSafety".DeselectBA40 := #unitInterface.specialFunctions.stack2InterfaceUnuse;
   "Safety.DataToSafety".DeselectBA15 := #unitInterface.specialFunctions.ReelCutBA015Unuse;
   "Safety.DataToSafety".DeselectBA60 := #unitInterface.specialFunctions.InspectionBA060Unuse;
END_REGION

REGION Network 46: Power On Command
   RUNG wire#powerrail
      Contact( #globalStatus.enablePower )
      Coil( "Safety.DataToSafety".PowerOnCommand )
   END_RUNG
   // the same network as SCL:
   "Safety.DataToSafety".PowerOnCommand := #globalStatus.enablePower;
END_REGION

REGION Network 47: OP Lamp
   RUNG wire#powerrail
      Contact( "Unit1.ControlNodes".InitializeEnable )
      Coil( "Safety.DataToSafety".OpLampStatus.InitializeEnable )
   END_RUNG
   RUNG wire#powerrail
      Contact( #statEmHomedCheck[0] )
      Coil( "Safety.DataToSafety".OpLampStatus.HomeLampStatus )
   END_RUNG
   // the same network as SCL:
   "Safety.DataToSafety".OpLampStatus.InitializeEnable := "Unit1.ControlNodes".InitializeEnable;
   "Safety.DataToSafety".OpLampStatus.HomeLampStatus := #statEmHomedCheck[0];
END_REGION

REGION Network 48: ScrapBox Status
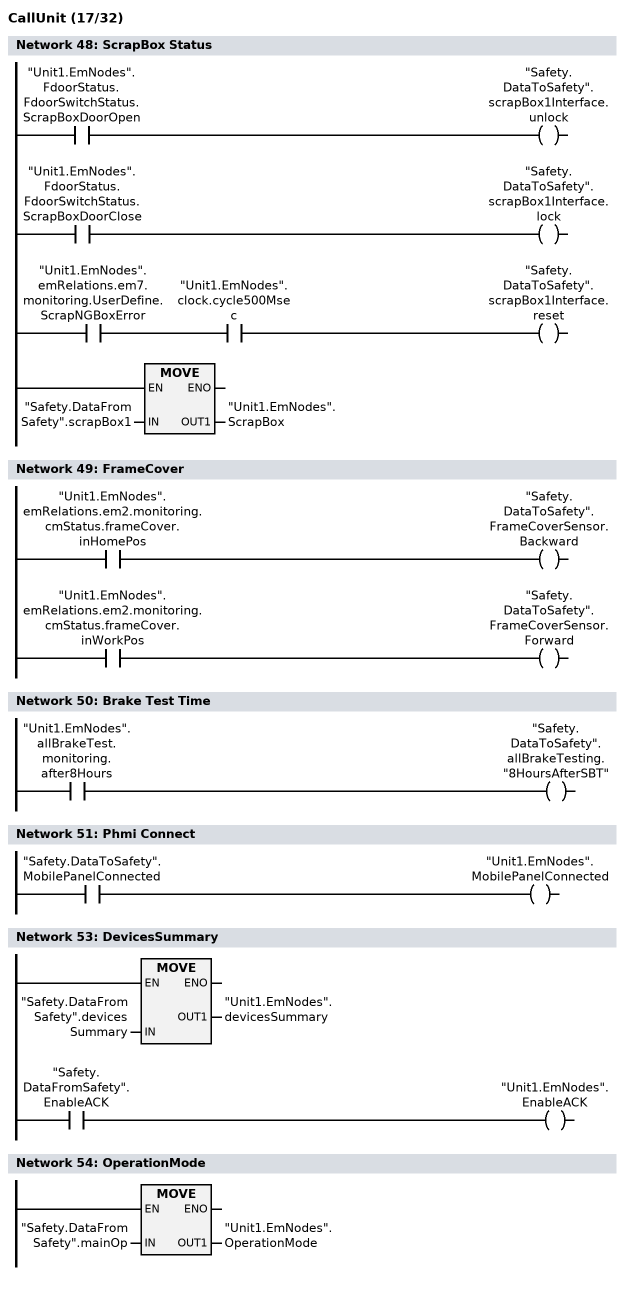
   RUNG wire#powerrail
      Contact( "Unit1.EmNodes".FdoorStatus.FdoorSwitchStatus.ScrapBoxDoorOpen )
      Coil( "Safety.DataToSafety".scrapBox1Interface.unlock )
   END_RUNG
   RUNG wire#powerrail
      Contact( "Unit1.EmNodes".FdoorStatus.FdoorSwitchStatus.ScrapBoxDoorClose )
      Coil( "Safety.DataToSafety".scrapBox1Interface.lock )
   END_RUNG
   RUNG wire#powerrail
      Contact( "Unit1.EmNodes".emRelations.em7.monitoring.UserDefine.ScrapNGBoxError )
      Contact( "Unit1.EmNodes".clock.cycle500Msec )
      Coil( "Safety.DataToSafety".scrapBox1Interface.reset )
   END_RUNG
   RUNG wire#powerrail
      Move(in := "Safety.DataFromSafety".scrapBox1, out1 => "Unit1.EmNodes".ScrapBox)
   END_RUNG
   // the same network as SCL:
   "Safety.DataToSafety".scrapBox1Interface.unlock := "Unit1.EmNodes".FdoorStatus.FdoorSwitchStatus.ScrapBoxDoorOpen;
   "Safety.DataToSafety".scrapBox1Interface.lock := "Unit1.EmNodes".FdoorStatus.FdoorSwitchStatus.ScrapBoxDoorClose;
   "Safety.DataToSafety".scrapBox1Interface.reset := "Unit1.EmNodes".emRelations.em7.monitoring.UserDefine.ScrapNGBoxError AND "Unit1.EmNodes".clock.cycle500Msec;
   "Unit1.EmNodes".ScrapBox := "Safety.DataFromSafety".scrapBox1;
END_REGION

REGION Network 49: FrameCover
   RUNG wire#powerrail
      Contact( "Unit1.EmNodes".emRelations.em2.monitoring.cmStatus.frameCover.inHomePos )
      Coil( "Safety.DataToSafety".FrameCoverSensor.Backward )
   END_RUNG
   RUNG wire#powerrail
      Contact( "Unit1.EmNodes".emRelations.em2.monitoring.cmStatus.frameCover.inWorkPos )
      Coil( "Safety.DataToSafety".FrameCoverSensor.Forward )
   END_RUNG
   // the same network as SCL:
   "Safety.DataToSafety".FrameCoverSensor.Backward := "Unit1.EmNodes".emRelations.em2.monitoring.cmStatus.frameCover.inHomePos;
   "Safety.DataToSafety".FrameCoverSensor.Forward := "Unit1.EmNodes".emRelations.em2.monitoring.cmStatus.frameCover.inWorkPos;
END_REGION

REGION Network 50: Brake Test Time
   RUNG wire#powerrail
      Contact( "Unit1.EmNodes".allBrakeTest.monitoring.after8Hours )
      Coil( "Safety.DataToSafety".allBrakeTesting."8HoursAfterSBT" )
   END_RUNG
   // the same network as SCL:
   "Safety.DataToSafety".allBrakeTesting."8HoursAfterSBT" := "Unit1.EmNodes".allBrakeTest.monitoring.after8Hours;
END_REGION

REGION Network 51: Phmi Connect
   RUNG wire#powerrail
      Contact( "Safety.DataToSafety".MobilePanelConnected )
      Coil( "Unit1.EmNodes".MobilePanelConnected )
   END_RUNG
   // the same network as SCL:
   "Unit1.EmNodes".MobilePanelConnected := "Safety.DataToSafety".MobilePanelConnected;
END_REGION

REGION Network 52: ******************** Data From Safety Mapping ********************
END_REGION

REGION Network 53: DevicesSummary
   RUNG wire#powerrail
      Move(in := "Safety.DataFromSafety".devicesSummary, out1 => "Unit1.EmNodes".devicesSummary)
   END_RUNG
   RUNG wire#powerrail
      Contact( "Safety.DataFromSafety".EnableACK )
      Coil( "Unit1.EmNodes".EnableACK )
   END_RUNG
   // the same network as SCL:
   "Unit1.EmNodes".devicesSummary := "Safety.DataFromSafety".devicesSummary;
   "Unit1.EmNodes".EnableACK := "Safety.DataFromSafety".EnableACK;
END_REGION

REGION Network 54: OperationMode
   RUNG wire#powerrail
      Move(in := "Safety.DataFromSafety".mainOp, out1 => "Unit1.EmNodes".OperationMode)
   END_RUNG
   // the same network as SCL:
   "Unit1.EmNodes".OperationMode := "Safety.DataFromSafety".mainOp;
END_REGION

REGION Network 55: PhmiMode
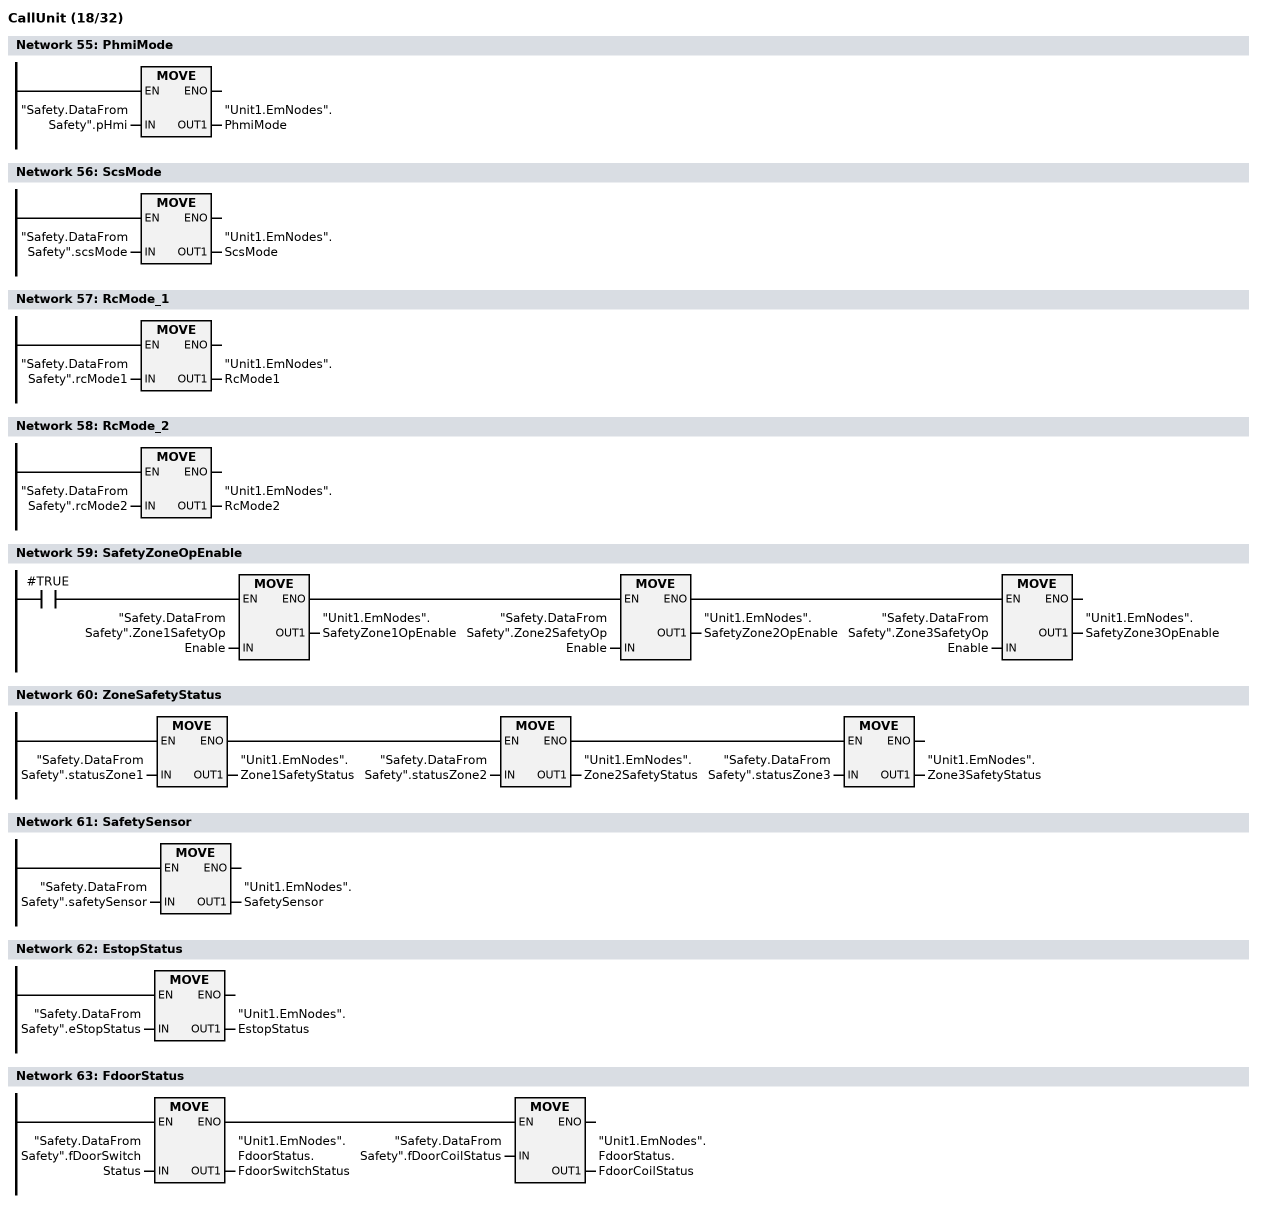
   RUNG wire#powerrail
      Move(in := "Safety.DataFromSafety".pHmi, out1 => "Unit1.EmNodes".PhmiMode)
   END_RUNG
   // the same network as SCL:
   "Unit1.EmNodes".PhmiMode := "Safety.DataFromSafety".pHmi;
END_REGION

REGION Network 56: ScsMode
   RUNG wire#powerrail
      Move(in := "Safety.DataFromSafety".scsMode, out1 => "Unit1.EmNodes".ScsMode)
   END_RUNG
   // the same network as SCL:
   "Unit1.EmNodes".ScsMode := "Safety.DataFromSafety".scsMode;
END_REGION

REGION Network 57: RcMode_1
   RUNG wire#powerrail
      Move(in := "Safety.DataFromSafety".rcMode1, out1 => "Unit1.EmNodes".RcMode1)
   END_RUNG
   // the same network as SCL:
   "Unit1.EmNodes".RcMode1 := "Safety.DataFromSafety".rcMode1;
END_REGION

REGION Network 58: RcMode_2
   RUNG wire#powerrail
      Move(in := "Safety.DataFromSafety".rcMode2, out1 => "Unit1.EmNodes".RcMode2)
   END_RUNG
   // the same network as SCL:
   "Unit1.EmNodes".RcMode2 := "Safety.DataFromSafety".rcMode2;
END_REGION

REGION Network 59: SafetyZoneOpEnable
   RUNG wire#powerrail
      Contact( #TRUE )
      Move(in := "Safety.DataFromSafety".Zone1SafetyOpEnable, out1 => "Unit1.EmNodes".SafetyZone1OpEnable)
      Move(in := "Safety.DataFromSafety".Zone2SafetyOpEnable, out1 => "Unit1.EmNodes".SafetyZone2OpEnable)
      Move(in := "Safety.DataFromSafety".Zone3SafetyOpEnable, out1 => "Unit1.EmNodes".SafetyZone3OpEnable)
   END_RUNG
   // the same network as SCL:
   IF #TRUE THEN
       "Unit1.EmNodes".SafetyZone1OpEnable := "Safety.DataFromSafety".Zone1SafetyOpEnable;
       "Unit1.EmNodes".SafetyZone2OpEnable := "Safety.DataFromSafety".Zone2SafetyOpEnable;
       "Unit1.EmNodes".SafetyZone3OpEnable := "Safety.DataFromSafety".Zone3SafetyOpEnable;
   END_IF;
END_REGION

REGION Network 60: ZoneSafetyStatus
   RUNG wire#powerrail
      Move(in := "Safety.DataFromSafety".statusZone1, out1 => "Unit1.EmNodes".Zone1SafetyStatus)
      Move(in := "Safety.DataFromSafety".statusZone2, out1 => "Unit1.EmNodes".Zone2SafetyStatus)
      Move(in := "Safety.DataFromSafety".statusZone3, out1 => "Unit1.EmNodes".Zone3SafetyStatus)
   END_RUNG
   // the same network as SCL:
   "Unit1.EmNodes".Zone1SafetyStatus := "Safety.DataFromSafety".statusZone1;
   "Unit1.EmNodes".Zone2SafetyStatus := "Safety.DataFromSafety".statusZone2;
   "Unit1.EmNodes".Zone3SafetyStatus := "Safety.DataFromSafety".statusZone3;
END_REGION

REGION Network 61: SafetySensor
   RUNG wire#powerrail
      Move(in := "Safety.DataFromSafety".safetySensor, out1 => "Unit1.EmNodes".SafetySensor)
   END_RUNG
   // the same network as SCL:
   "Unit1.EmNodes".SafetySensor := "Safety.DataFromSafety".safetySensor;
END_REGION

REGION Network 62: EstopStatus
   RUNG wire#powerrail
      Move(in := "Safety.DataFromSafety".eStopStatus, out1 => "Unit1.EmNodes".EstopStatus)
   END_RUNG
   // the same network as SCL:
   "Unit1.EmNodes".EstopStatus := "Safety.DataFromSafety".eStopStatus;
END_REGION

REGION Network 63: FdoorStatus
   RUNG wire#powerrail
      Move(in := "Safety.DataFromSafety".fDoorSwitchStatus, out1 => "Unit1.EmNodes".FdoorStatus.FdoorSwitchStatus)
      Move(in := "Safety.DataFromSafety".fDoorCoilStatus, out1 => "Unit1.EmNodes".FdoorStatus.FdoorCoilStatus)
   END_RUNG
   // the same network as SCL:
   "Unit1.EmNodes".FdoorStatus.FdoorSwitchStatus := "Safety.DataFromSafety".fDoorSwitchStatus;
   "Unit1.EmNodes".FdoorStatus.FdoorCoilStatus := "Safety.DataFromSafety".fDoorCoilStatus;
END_REGION

REGION Network 64: Roll Change Mode Active
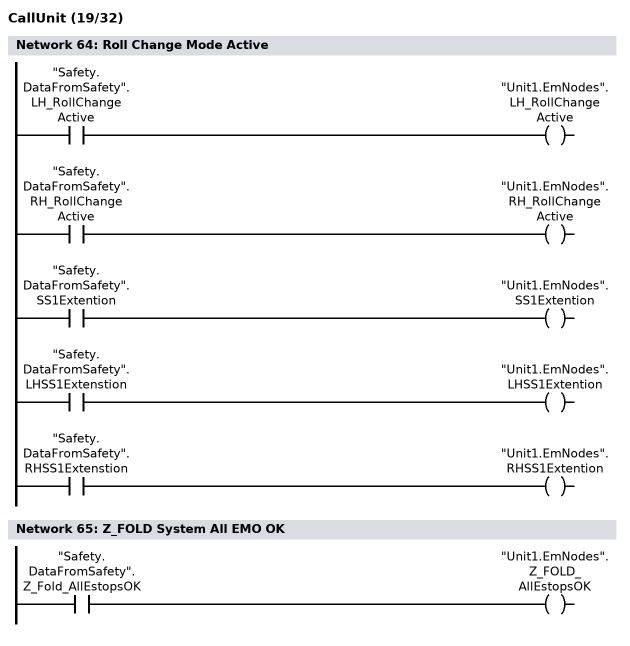
   RUNG wire#powerrail
      Contact( "Safety.DataFromSafety".LH_RollChangeActive )
      Coil( "Unit1.EmNodes".LH_RollChangeActive )
   END_RUNG
   RUNG wire#powerrail
      Contact( "Safety.DataFromSafety".RH_RollChangeActive )
      Coil( "Unit1.EmNodes".RH_RollChangeActive )
   END_RUNG
   RUNG wire#powerrail
      Contact( "Safety.DataFromSafety".SS1Extention )
      Coil( "Unit1.EmNodes".SS1Extention )
   END_RUNG
   RUNG wire#powerrail
      Contact( "Safety.DataFromSafety".LHSS1Extenstion )
      Coil( "Unit1.EmNodes".LHSS1Extention )
   END_RUNG
   RUNG wire#powerrail
      Contact( "Safety.DataFromSafety".RHSS1Extenstion )
      Coil( "Unit1.EmNodes".RHSS1Extention )
   END_RUNG
   // the same network as SCL:
   "Unit1.EmNodes".LH_RollChangeActive := "Safety.DataFromSafety".LH_RollChangeActive;
   "Unit1.EmNodes".RH_RollChangeActive := "Safety.DataFromSafety".RH_RollChangeActive;
   "Unit1.EmNodes".SS1Extention := "Safety.DataFromSafety".SS1Extention;
   "Unit1.EmNodes".LHSS1Extention := "Safety.DataFromSafety".LHSS1Extenstion;
   "Unit1.EmNodes".RHSS1Extention := "Safety.DataFromSafety".RHSS1Extenstion;
END_REGION

REGION Network 65: Z_FOLD System All EMO OK
   RUNG wire#powerrail
      Contact( "Safety.DataFromSafety".Z_Fold_AllEstopsOK )
      Coil( "Unit1.EmNodes".Z_FOLD_AllEstopsOK )
   END_RUNG
   // the same network as SCL:
   "Unit1.EmNodes".Z_FOLD_AllEstopsOK := "Safety.DataFromSafety".Z_Fold_AllEstopsOK;
END_REGION

REGION Network 66: ******************** FAT Mode ********************
END_REGION

